# B&R Automation Studio project NAELD004C00R10L518F00 (part 32)

#### Act_Main.st
```iecst
(** 2019-10-30 **)
ACTION Act_Main:

	IF eStatOld <> eStat THEN
		fbInit(bEn := FALSE);
		fbEnt(bEn := FALSE);
		fbPreExit(bEn := FALSE);
		fbExit(bEn := FALSE);
		fbExit1(bEn := FALSE);
		fbStop(bEn := FALSE);
		fbFixClprClampChk(bEn := FALSE);
		fbFixClprUnclampChk(bEn := FALSE);
		fbRmtClprClampChk(bEn := FALSE);
		fbRmtClprUnclampChk(bEn := FALSE);
		fbClprDlyTm(IN := FALSE);

		IF eStatOld <> MagConv2ClpActIdle
			AND eStatOld <> MagConv2ClpActSetMtrSigOnOrLToR
			AND eStatOld <> MagConv2ClpActSetMtrDirOrRToL
			AND eStatOld <> MagConv2ClpActRstMtrSigOnOrLToR
			AND eStatOld <> MagConv2ClpActRstMtrDirOrRToL
			AND eStatOld <> MagConv2ClpActSetMtrAll
			AND eStatOld <> MagConv2ClpActRstMtrAll THEN

			bMtrSigOnOrLToR	:= FALSE;
			bMtrDirOrRToL	:= FALSE;

		END_IF

		usiStep		:= 0;
		usiSubStep	:= 0;
		bReachEnd	:= FALSE;

		sStatTxt	:= a_sStatText[eStat];

		eStatOld	:= eStat;

		eStatus		:= Busy;
	END_IF

	//Main
	CASE eStat OF

		MagConv2ClpActIdle:
			IF EDGENEG(p_bManual) THEN
				bMtrSigOnOrLToR	:= FALSE;
				bMtrDirOrRToL	:= FALSE;
			END_IF

			eStatus	:= Idle;

		MagConv2ClpActInit:
			IF eStatus = Idle OR eStatus = Busy THEN

				eStatus	:= Busy;

				//Magazine Conveyor Init Run
				//Detect Have Magazine
				IF p_bLeftSen OR p_bRightSen THEN
					bHvMag	:= TRUE;
				ELSE
					bHvMag	:= FALSE;
				END_IF

				fbInit.bConvLToR	:= (p_eDirection = ConvDirLToR) OR (p_eDirection = ConvDirLToL);
				fbInit.tTxDlyTm		:= DINT_TO_TIME(p_diInitTm);

				IF fbInit.bConvLToR = TRUE THEN
					fbInit.bEndSen	:= p_bRightSen;
				ELSE
					fbInit.bEndSen	:= p_bLeftSen;
				END_IF

				fbInit(bEn := TRUE);

				bMtrSigOnOrLToR	:= fbInit.bMtrSigOnOrLToR;
				bMtrDirOrRToL	:= fbInit.bMtrDirOrRToL;

				IF fbInit.udiStatus = 0 THEN
					IF fbInit.bConvLToR = TRUE THEN
						IF bHvMag = TRUE AND p_bRightSen = FALSE THEN
							udiStatus	:= 10000;	//Magazine Detected But Not Present At Outlet Sensor (L - R) While Magazine Conveyor Initial
							eStatus		:= Error;
						ELSE
							eStatus	:= Done;
						END_IF
					ELSE
						IF bHvMag = TRUE AND p_bLeftSen = FALSE THEN
							udiStatus	:= 10001;	//Magazine Detected But Not Present At Outlet Sensor (R - L) While Magazine Conveyor Initial
							eStatus		:= Error;
						ELSE
							eStatus	:= Done;
						END_IF
					END_IF
				ELSIF fbInit.udiStatus < 65534 THEN
					udiStatus	:= fbInit.udiStatus;
					eStatus		:= Error;
				END_IF
			END_IF

		MagConv2ClpActInitStopClp:
			IF eStatus = Idle OR eStatus = Busy THEN

				eStatus	:= Busy;

				CASE usiStep OF
					0:	//Unclamp
						bFixClprClampCtrl	:= FALSE;
						bRmtClprClampCtrl	:= FALSE;

						fbFixClprUnclampChk.bExtSen		:= p_bFixClprClampSen;
						fbFixClprUnclampChk.bRetSen		:= p_bFixClprUnclampSen;
						fbFixClprUnclampChk.bRetSafety	:= p_bFixClprUnclampSafetySen;
						fbFixClprUnclampChk(bEn := TRUE);

						fbRmtClprUnclampChk.bExtSen		:= p_bRmtClprClampSen;
						fbRmtClprUnclampChk.bRetSen		:= p_bRmtClprUnclampSen;
						fbRmtClprUnclampChk.bRetSafety	:= p_bRmtClprUnclampSafetySen;
						fbRmtClprUnclampChk(bEn := TRUE);

						IF fbFixClprUnclampChk.udiStatus = 0 AND fbRmtClprUnclampChk.udiStatus = 0 THEN
							usiStep	:= 1;
						ELSIF (fbFixClprUnclampChk.udiStatus > 0 AND fbFixClprUnclampChk.udiStatus < 65534) OR (fbRmtClprUnclampChk.udiStatus > 0 AND fbRmtClprUnclampChk.udiStatus < 65534) THEN
							bFixClprClampCtrl	:= TRUE;
							bRmtClprClampCtrl	:= TRUE;

							eStatus	:= Error;

							IF fbFixClprUnclampChk.udiStatus = 1504 OR fbRmtClprUnclampChk.udiStatus = 1504 THEN
								udiStatus	:= 10002;	//Clamper Clamp Sensor Off Time Out In Unclamp Check While Conveyor Initial With Clamper
							ELSIF fbFixClprUnclampChk.udiStatus = 1505 OR fbRmtClprUnclampChk.udiStatus = 1505 THEN
								udiStatus	:= 10003;	//Clamper Unclamp Sensor On Time Out In Unclamp Check While Conveyor Initial With Clamper
							ELSIF fbFixClprUnclampChk.udiStatus = 1508 OR fbRmtClprUnclampChk.udiStatus = 1508 THEN
								udiStatus	:= 10004;	//Clamper Unclamp Safety Sensor Error In Unclamp Check While Conveyor Initial With Clamper
							ELSE
								IF fbFixClprUnclampChk.udiStatus > 0 AND fbFixClprUnclampChk.udiStatus < 65534 THEN
									udiStatus	:= fbFixClprUnclampChk.udiStatus;
								ELSIF fbRmtClprUnclampChk.udiStatus > 0 AND fbRmtClprUnclampChk.udiStatus < 65534 THEN
									udiStatus	:= fbRmtClprUnclampChk.udiStatus;
								END_IF
							END_IF
						END_IF

					1:	//Magazine Conveyor Init Run
						//Detect Have Magazine
						IF p_bLeftSen OR p_bRightSen THEN
							bHvMag	:= TRUE;
						ELSE
							bHvMag	:= FALSE;
						END_IF

						fbInit.bConvLToR	:= (p_eDirection = ConvDirLToR) OR (p_eDirection = ConvDirLToL);
						fbInit.tTxDlyTm		:= DINT_TO_TIME(p_diInitTm);

						IF fbInit.bConvLToR = TRUE THEN
							fbInit.bEndSen	:= p_bRightSen;
						ELSE
							fbInit.bEndSen	:= p_bLeftSen;
						END_IF

						fbInit(bEn := TRUE);

						bMtrSigOnOrLToR	:= fbInit.bMtrSigOnOrLToR;
						bMtrDirOrRToL	:= fbInit.bMtrDirOrRToL;

						IF fbInit.udiStatus = 0 THEN
							IF fbInit.bConvLToR = TRUE THEN
								IF bHvMag = TRUE AND p_bRightSen = FALSE THEN
									udiStatus	:= 10005;	//Magazine Detected But Not Present At Outlet Sensor (L - R) While Conveyor Initial With Clamper
									eStatus		:= Error;
								ELSE
									usiStep	:= 2;
								END_IF
							ELSE
								IF bHvMag = TRUE AND p_bLeftSen = FALSE THEN
									udiStatus	:= 10006;	//Magazine Detected But Not Present At Outlet Sensor (R - L) While Conveyor Initial With Clamper
									eStatus		:= Error;
								ELSE
									usiStep	:= 2;
								END_IF
							END_IF
						ELSIF fbInit.udiStatus < 65534 THEN
							udiStatus	:= fbInit.udiStatus;
							eStatus		:= Error;
						END_IF

					2:	//Check If Have Magazine
						IF bHvMag = TRUE THEN
							usiStep	:= 4;
						ELSE
							eStatus	:= Done;
						END_IF

					3:	//Fix Clamp
						bFixClprClampCtrl	:= TRUE;

						fbFixClprClampChk.bExtSen		:= p_bFixClprClampSen;
						fbFixClprClampChk.bRetSen		:= p_bFixClprUnclampSen;
						fbFixClprClampChk.bExtSafety	:= p_bFixClprClampSafetySen;
						fbFixClprClampChk(bEn := TRUE);

						IF fbFixClprClampChk.udiStatus = 0 THEN
							//	usiStep	:= 4;
							eStatus	:= Done;
						ELSIF fbFixClprClampChk.udiStatus < 65534 THEN
							bFixClprClampCtrl	:= FALSE;

							eStatus	:= Error;

							IF fbFixClprClampChk.udiStatus = 1503 THEN
								udiStatus	:= 10007;	//Clamper Clamp Sensor On Time Out In Clamp Check While Conveyor Initial With Clamper
							ELSIF fbFixClprClampChk.udiStatus = 1506 THEN
								udiStatus	:= 10008;	//Clamper Unclamp Sensor Off Time Out In Clamp Check While Conveyor Initial With Clamper
							ELSIF fbFixClprClampChk.udiStatus = 1507 THEN
								udiStatus	:= 10009;	//Clamper Clamp Safety Sensor Error In Clamp Check While Conveyor Initial With Clamper
							ELSE
								udiStatus	:= fbFixClprClampChk.udiStatus;
							END_IF
						END_IF

					4:	//Remote Clamp
						bRmtClprClampCtrl	:= TRUE;

						fbRmtClprClampChk.bExtSen		:= p_bRmtClprClampSen;
						fbRmtClprClampChk.bRetSen		:= p_bRmtClprUnclampSen;
						fbRmtClprClampChk.bExtSafety	:= p_bRmtClprClampSafetySen;
						fbRmtClprClampChk(bEn := TRUE);

						IF fbRmtClprClampChk.udiStatus = 0 THEN
							//	eStatus	:= Done;
							usiStep	:= 3;
						ELSIF fbRmtClprClampChk.udiStatus < 65534 THEN
							bRmtClprClampCtrl	:= FALSE;

							eStatus	:= Error;

							IF fbRmtClprClampChk.udiStatus = 1503 THEN
								udiStatus	:= 10007;	//Clamper Clamp Sensor On Time Out In Clamp Check While Conveyor Initial With Clamper
							ELSIF fbRmtClprClampChk.udiStatus = 1506 THEN
								udiStatus	:= 10008;	//Clamper Unclamp Sensor Off Time Out In Clamp Check While Conveyor Initial With Clamper
							ELSIF fbRmtClprClampChk.udiStatus = 1507 THEN
								udiStatus	:= 10009;	//Clamper Clamp Safety Sensor Error In Clamp Check While Conveyor Initial With Clamper
							ELSE
								udiStatus	:= fbRmtClprClampChk.udiStatus;
							END_IF
						END_IF

				END_CASE
			END_IF

		MagConv2ClpActInitClpStop:
			IF eStatus = Idle OR eStatus = Busy THEN

				eStatus	:= Busy;

				CASE usiStep OF
					0:	//Unclamp
						bFixClprClampCtrl	:= FALSE;
						bRmtClprClampCtrl	:= FALSE;

						fbFixClprUnclampChk.bExtSen		:= p_bFixClprClampSen;
						fbFixClprUnclampChk.bRetSen		:= p_bFixClprUnclampSen;
						fbFixClprUnclampChk.bRetSafety	:= p_bFixClprUnclampSafetySen;
						fbFixClprUnclampChk(bEn := TRUE);

						fbRmtClprUnclampChk.bExtSen		:= p_bRmtClprClampSen;
						fbRmtClprUnclampChk.bRetSen		:= p_bRmtClprUnclampSen;
						fbRmtClprUnclampChk.bRetSafety	:= p_bRmtClprUnclampSafetySen;
						fbRmtClprUnclampChk(bEn := TRUE);

						IF fbFixClprUnclampChk.udiStatus = 0 AND fbRmtClprUnclampChk.udiStatus = 0 THEN
							usiStep	:= 1;
						ELSIF (fbFixClprUnclampChk.udiStatus > 0 AND fbFixClprUnclampChk.udiStatus < 65534) OR (fbRmtClprUnclampChk.udiStatus > 0 AND fbRmtClprUnclampChk.udiStatus < 65534) THEN
							bFixClprClampCtrl	:= TRUE;
							bRmtClprClampCtrl	:= TRUE;

							eStatus	:= Error;

							IF fbFixClprUnclampChk.udiStatus = 1504 OR fbRmtClprUnclampChk.udiStatus = 1504 THEN
								udiStatus	:= 10002;	//Clamper Clamp Sensor Off Time Out In Unclamp Check While Conveyor Initial With Clamper
							ELSIF fbFixClprUnclampChk.udiStatus = 1505 OR fbRmtClprUnclampChk.udiStatus = 1505 THEN
								udiStatus	:= 10003;	//Clamper Unclamp Sensor On Time Out In Unclamp Check While Conveyor Initial With Clamper
							ELSIF fbFixClprUnclampChk.udiStatus = 1508 OR fbRmtClprUnclampChk.udiStatus = 1508 THEN
								udiStatus	:= 10004;	//Clamper Unclamp Safety Sensor Error In Unclamp Check While Conveyor Initial With Clamper
							ELSE
								IF fbFixClprUnclampChk.udiStatus > 0 AND fbFixClprUnclampChk.udiStatus < 65534 THEN
									udiStatus	:= fbFixClprUnclampChk.udiStatus;
								ELSIF fbRmtClprUnclampChk.udiStatus > 0 AND fbRmtClprUnclampChk.udiStatus < 65534 THEN
									udiStatus	:= fbRmtClprUnclampChk.udiStatus;
								END_IF
							END_IF
						END_IF

					1:	//Magazine Conveyor Init Run & Clamp
						//Detect Have Magazine
						IF p_bLeftSen OR p_bRightSen THEN
							bHvMag	:= TRUE;
						ELSE
							bHvMag	:= FALSE;
						END_IF

						fbInit.bConvLToR	:= (p_eDirection = ConvDirLToR) OR (p_eDirection = ConvDirLToL);
						fbInit.tTxDlyTm		:= DINT_TO_TIME(p_diInitTm);

						IF fbInit.bConvLToR = TRUE THEN
							fbInit.bEndSen	:= p_bRightSen;
						ELSE
							fbInit.bEndSen	:= p_bLeftSen;
						END_IF

						fbInit(bEn := TRUE);

						bMtrSigOnOrLToR	:= fbInit.bMtrSigOnOrLToR;
						bMtrDirOrRToL	:= fbInit.bMtrDirOrRToL;

						IF fbInit.bEndSen = TRUE THEN
							bReachEnd	:= TRUE;
						END_IF

						IF bReachEnd = TRUE THEN
							fbClprDlyTm(IN := TRUE);
							IF fbClprDlyTm.Q = TRUE THEN
								CASE usiSubStep OF
									//	0:	//Fix Clamp
									//										bFixClprClampCtrl	:= TRUE;

									//										fbFixClprClampChk.bExtSen		:= p_bFixClprClampSen;
									//										fbFixClprClampChk.bRetSen		:= p_bFixClprUnclampSen;
									//										fbFixClprClampChk.bExtSafety	:= p_bFixClprClampSafetySen;
									//										fbFixClprClampChk(bEn := TRUE);
									//
									//										IF fbFixClprClampChk.udiStatus = 0 THEN
									//											usiSubStep	:= 1;
									//										END_IF

									0:	//Remote Clamp
										bRmtClprClampCtrl	:= TRUE;

										fbRmtClprClampChk.bExtSen		:= p_bRmtClprClampSen;
										fbRmtClprClampChk.bRetSen		:= p_bRmtClprUnclampSen;
										fbRmtClprClampChk.bExtSafety	:= p_bRmtClprClampSafetySen;
										fbRmtClprClampChk(bEn := TRUE);

										IF fbRmtClprClampChk.udiStatus = 0 THEN
											usiSubStep	:= 1;
										END_IF

									1:

										bFixClprClampCtrl	:= TRUE;

										fbFixClprClampChk.bExtSen		:= p_bFixClprClampSen;
										fbFixClprClampChk.bRetSen		:= p_bFixClprUnclampSen;
										fbFixClprClampChk.bExtSafety	:= p_bFixClprClampSafetySen;
										fbFixClprClampChk(bEn := TRUE);

								END_CASE
							END_IF
						END_IF

						IF (fbInit.udiStatus = 0) AND ((fbFixClprClampChk.udiStatus = 0 AND fbRmtClprClampChk.udiStatus = 0) OR (bReachEnd = FALSE)) THEN
							IF fbInit.bConvLToR = TRUE THEN
								IF bHvMag = TRUE AND p_bRightSen = FALSE THEN
									udiStatus	:= 10041;	//Magazine Detected But Not Present At Outlet Sensor (L - R) While Conveyor Initial With Clamper
									eStatus		:= Error;
								ELSE
									eStatus		:= Done;
								END_IF
							ELSE
								IF bHvMag = TRUE AND p_bLeftSen = FALSE THEN
									udiStatus	:= 10042;	//Magazine Detected But Not Present At Outlet Sensor (R - L) While Conveyor Initial With Clamper
									eStatus		:= Error;
								ELSE
									eStatus		:= Done;
								END_IF
							END_IF

						ELSIF fbInit.udiStatus > 0 AND fbInit.udiStatus < 65534 THEN
							udiStatus	:= fbInit.udiStatus;
							eStatus		:= Error;

						ELSIF (fbFixClprClampChk.udiStatus > 0 AND fbFixClprClampChk.udiStatus < 65534) OR (fbRmtClprClampChk.udiStatus > 0 AND fbRmtClprClampChk.udiStatus < 65534) THEN
							bFixClprClampCtrl	:= FALSE;
							bRmtClprClampCtrl	:= FALSE;

							eStatus	:= Error;

							IF fbFixClprClampChk.udiStatus = 1503 OR fbRmtClprClampChk.udiStatus = 1503 THEN
								udiStatus	:= 10043;	//Clamper Clamp Sensor On Time Out In Clamp Check While Conveyor Initial With Clamper
							ELSIF fbFixClprClampChk.udiStatus = 1506 OR fbRmtClprClampChk.udiStatus = 1506 THEN
								udiStatus	:= 10044;	//Clamper Unclamp Sensor Off Time Out In Clamp Check While Conveyor Initial With Clamper
							ELSIF fbFixClprClampChk.udiStatus = 1507 OR fbRmtClprClampChk.udiStatus = 1507 THEN
								udiStatus	:= 10045;	//Clamper Clamp Safety Sensor Error In Clamp Check While Conveyor Initial With Clamper
							ELSE
								IF fbFixClprClampChk.udiStatus > 0 AND fbFixClprClampChk.udiStatus < 65534 THEN
									udiStatus	:= fbFixClprClampChk.udiStatus;
								ELSIF fbRmtClprClampChk.udiStatus > 0 AND fbRmtClprClampChk.udiStatus < 65534 THEN
									udiStatus	:= fbRmtClprClampChk.udiStatus;
								END_IF
							END_IF
						END_IF

				END_CASE
			END_IF

		MagConv2ClpActEnt:
			IF eStatus = Idle OR eStatus = Busy THEN

				eStatus	:= Busy;

				//Detect Have Magazine
				IF p_bLeftSen OR p_bRightSen THEN
					bHvMag	:= TRUE;
				END_IF

				//Conveyor Run
				fbEnt.bConvLToR		:= (p_eDirection = ConvDirLToR) OR (p_eDirection = ConvDirLToL);
				fbEnt.tTimeOut		:= DINT_TO_TIME(p_diTxInTimeOut);

				IF fbEnt.bConvLToR = TRUE THEN
					fbEnt.bEndSen	:= p_bRightSen;
				ELSE
					fbEnt.bEndSen	:= p_bLeftSen;
				END_IF

				fbEnt(bEn := TRUE);

				bMtrSigOnOrLToR	:= fbEnt.bMtrSigOnOrLToR;
				bMtrDirOrRToL	:= fbEnt.bMtrDirOrRToL;

				IF fbEnt.udiStatus = 0 THEN
					eStatus		:= Done;
				ELSIF fbEnt.udiStatus < 65534 THEN
					eStatus		:= Error;

					IF fbEnt.udiStatus = 1101 THEN
						udiStatus	:= 10028;	//Transfer In Time Out While Entering Magazine
					ELSE
						udiStatus	:= fbEnt.udiStatus;
					END_IF
				END_IF

			END_IF

		MagConv2ClpActEntStopClp:
			IF eStatus = Idle OR eStatus = Busy THEN

				eStatus	:= Busy;

				CASE usiStep OF
					0:	//Conveyor Enter
						//Detect Have Magazine
						IF p_bLeftSen OR p_bRightSen THEN
							bHvMag	:= TRUE;
						END_IF

						//Conveyor Run
						fbEnt.bConvLToR		:= (p_eDirection = ConvDirLToR) OR (p_eDirection = ConvDirLToL);
						fbEnt.tTimeOut		:= DINT_TO_TIME(p_diTxInTimeOut);

						IF fbEnt.bConvLToR = TRUE THEN
							fbEnt.bEndSen	:= p_bRightSen;
						ELSE
							fbEnt.bEndSen	:= p_bLeftSen;
						END_IF

						fbEnt(bEn := TRUE);

						bMtrSigOnOrLToR	:= fbEnt.bMtrSigOnOrLToR;
						bMtrDirOrRToL	:= fbEnt.bMtrDirOrRToL;

						IF fbEnt.udiStatus = 0 THEN
							usiStep	:= 2;
						ELSIF fbEnt.udiStatus < 65534 THEN
							eStatus	:= Error;

							IF fbEnt.udiStatus = 1101 THEN
								udiStatus	:= 10029;	//Transfer In Time Out While Entering Magazine
							ELSE
								udiStatus	:= fbEnt.udiStatus;
							END_IF
						END_IF

					1:	//Fix Clamp
						bFixClprClampCtrl	:= TRUE;

						fbFixClprClampChk.bExtSen		:= p_bFixClprClampSen;
						fbFixClprClampChk.bRetSen		:= p_bFixClprUnclampSen;
						fbFixClprClampChk.bExtSafety	:= p_bFixClprClampSafetySen;
						fbFixClprClampChk(bEn := TRUE);

						IF fbFixClprClampChk.udiStatus = 0 THEN
							//usiStep	:= 2;
							eStatus	:= Done;
						ELSIF fbFixClprClampChk.udiStatus < 65534 THEN
							bFixClprClampCtrl	:= FALSE;

							eStatus	:= Error;

							IF fbFixClprClampChk.udiStatus = 1503 THEN
								udiStatus	:= 10010;	//Clamper Clamp Sensor On Time Out In Clamp Check While Conveyor Enter With Clamper
							ELSIF fbFixClprClampChk.udiStatus = 1506 THEN
								udiStatus	:= 10011;	//Clamper Unclamp Sensor Off Time Out In Clamp Check While Conveyor Enter With Clamper
							ELSIF fbFixClprClampChk.udiStatus = 1507 THEN
								udiStatus	:= 10012;	//Clamper Clamp Safety Sensor Error In Clamp Check While Conveyor Enter With Clamper
							ELSE
								udiStatus	:= fbFixClprClampChk.udiStatus;
							END_IF
						END_IF

					2:	//Remote Clamp
						bRmtClprClampCtrl	:= TRUE;

						fbRmtClprClampChk.bExtSen		:= p_bRmtClprClampSen;
						fbRmtClprClampChk.bRetSen		:= p_bRmtClprUnclampSen;
						fbRmtClprClampChk.bExtSafety	:= p_bRmtClprClampSafetySen;
						fbRmtClprClampChk(bEn := TRUE);

						IF fbRmtClprClampChk.udiStatus = 0 THEN
							//	eStatus	:= Done;
							usiStep	:= 1;
						ELSIF fbRmtClprClampChk.udiStatus < 65534 THEN
							bRmtClprClampCtrl	:= FALSE;

							eStatus	:= Error;

							IF fbRmtClprClampChk.udiStatus = 1503 THEN
								udiStatus	:= 10010;	//Clamper Clamp Sensor On Time Out In Clamp Check While Conveyor Enter With Clamper
							ELSIF fbRmtClprClampChk.udiStatus = 1506 THEN
								udiStatus	:= 10011;	//Clamper Unclamp Sensor Off Time Out In Clamp Check While Conveyor Enter With Clamper
							ELSIF fbRmtClprClampChk.udiStatus = 1507 THEN
								udiStatus	:= 10012;	//Clamper Clamp Safety Sensor Error In Clamp Check While Conveyor Enter With Clamper
							ELSE
								udiStatus	:= fbRmtClprClampChk.udiStatus;
							END_IF
						END_IF

				END_CASE

			END_IF

		MagConv2ClpActEntClpStop:
			IF eStatus = Idle OR eStatus = Busy THEN

				eStatus	:= Busy;

				//Detect Have Magazine
				IF p_bLeftSen OR p_bRightSen THEN
					bHvMag	:= TRUE;
				END_IF

				//Conveyor Run
				fbEnt.bConvLToR		:= (p_eDirection = ConvDirLToR) OR (p_eDirection = ConvDirLToL);
				fbEnt.tTimeOut		:= DINT_TO_TIME(p_diTxInTimeOut);

				IF fbEnt.bConvLToR = TRUE THEN
					fbEnt.bEndSen	:= p_bRightSen;
				ELSE
					fbEnt.bEndSen	:= p_bLeftSen;
				END_IF

				fbEnt(bEn := TRUE);

				bMtrSigOnOrLToR	:= fbEnt.bMtrSigOnOrLToR;
				bMtrDirOrRToL	:= fbEnt.bMtrDirOrRToL;

				IF fbEnt.bEndSen = TRUE THEN
					bReachEnd	:= TRUE;
				END_IF

				IF bReachEnd = TRUE THEN
					fbClprDlyTm(IN := TRUE);
					IF fbClprDlyTm.Q = TRUE THEN
						CASE usiSubStep OF
							0:	//Fix Clamp
								//								bFixClprClampCtrl	:= TRUE;
								//
								//								fbFixClprClampChk.bExtSen		:= p_bFixClprClampSen;
								//								fbFixClprClampChk.bRetSen		:= p_bFixClprUnclampSen;
								//								fbFixClprClampChk.bExtSafety	:= p_bFixClprClampSafetySen;
								//								fbFixClprClampChk(bEn := TRUE);
								//
								//								IF fbFixClprClampChk.udiStatus = 0 THEN
								//									usiSubStep	:= 1;
								//								END_IF

								bRmtClprClampCtrl	:= TRUE;

								fbRmtClprClampChk.bExtSen		:= p_bRmtClprClampSen;
								fbRmtClprClampChk.bRetSen		:= p_bRmtClprUnclampSen;
								fbRmtClprClampChk.bExtSafety	:= p_bRmtClprClampSafetySen;
								fbRmtClprClampChk(bEn := TRUE);

								IF fbRmtClprClampChk.udiStatus = 0 THEN
									usiSubStep	:= 1;
								END_IF

							1:	//Remote Clamp
								//								bRmtClprClampCtrl	:= TRUE;
								//
								//								fbRmtClprClampChk.bExtSen		:= p_bRmtClprClampSen;
								//								fbRmtClprClampChk.bRetSen		:= p_bRmtClprUnclampSen;
								//								fbRmtClprClampChk.bExtSafety	:= p_bRmtClprClampSafetySen;
								//								fbRmtClprClampChk(bEn := TRUE);

								bFixClprClampCtrl	:= TRUE;

								fbFixClprClampChk.bExtSen		:= p_bFixClprClampSen;
								fbFixClprClampChk.bRetSen		:= p_bFixClprUnclampSen;
								fbFixClprClampChk.bExtSafety	:= p_bFixClprClampSafetySen;
								fbFixClprClampChk(bEn := TRUE);

						END_CASE
					END_IF
				END_IF

				IF fbEnt.udiStatus = 0 AND (fbFixClprClampChk.udiStatus = 0 AND fbRmtClprClampChk.udiStatus = 0) THEN
					eStatus	:= Done;

				ELSIF (fbFixClprClampChk.udiStatus > 0 AND fbFixClprClampChk.udiStatus < 65534) OR (fbRmtClprClampChk.udiStatus > 0 AND fbRmtClprClampChk.udiStatus < 65534) THEN
					bFixClprClampCtrl	:= FALSE;
					bRmtClprClampCtrl	:= FALSE;

					eStatus	:= Error;

					IF fbFixClprClampChk.udiStatus = 1503 OR fbRmtClprClampChk.udiStatus = 1503 THEN
						udiStatus	:= 10034;	//Clamper Clamp Sensor On Time Out In Clamp Check While Conveyor Enter With Clamper
					ELSIF fbFixClprClampChk.udiStatus = 1506 OR fbRmtClprClampChk.udiStatus = 1506 THEN
						udiStatus	:= 10035;	//Clamper Unclamp Sensor Off Time Out In Clamp Check While Conveyor Enter With Clamper
					ELSIF fbFixClprClampChk.udiStatus = 1507 OR fbRmtClprClampChk.udiStatus = 1507 THEN
						udiStatus	:= 10036;	//Clamper Clamp Safety Sensor Error In Clamp Check While Conveyor Enter With Clamper
					ELSE
						IF fbFixClprClampChk.udiStatus > 0 AND fbFixClprClampChk.udiStatus < 65534 THEN
							udiStatus	:= fbFixClprClampChk.udiStatus;
						ELSIF fbRmtClprClampChk.udiStatus > 0 AND fbRmtClprClampChk.udiStatus < 65534 THEN
							udiStatus	:= fbRmtClprClampChk.udiStatus;
						END_IF
					END_IF

				ELSIF fbEnt.udiStatus > 0 AND fbEnt.udiStatus < 65534 THEN
					eStatus	:= Error;

					IF fbEnt.udiStatus = 1101 THEN
						udiStatus	:= 10037;	//Transfer In Time Out While Entering Magazine
					ELSE
						udiStatus	:= fbEnt.udiStatus;
					END_IF

				END_IF

			END_IF

		MagConv2ClpActPreExit:
			IF eStatus = Idle OR eStatus = Busy THEN

				eStatus	:= Busy;

				//Conveyor Run
				fbPreExit.bConvLToR		:= (p_eDirection = ConvDirLToR) OR (p_eDirection = ConvDirRToR);
				fbPreExit.tTxDlyTm		:= DINT_TO_TIME(p_diInitTm);

				IF fbPreExit.bConvLToR = TRUE THEN
					fbPreExit.bEndSen	:= p_bRightSen;
					fbPreExit.bStartSen	:= p_bLeftSen;
				ELSE
					fbPreExit.bEndSen	:= p_bLeftSen;
					fbPreExit.bStartSen	:= p_bRightSen;
				END_IF

				fbPreExit(bEn := TRUE);

				bMtrSigOnOrLToR	:= fbPreExit.bMtrSigOnOrLToR;
				bMtrDirOrRToL	:= fbPreExit.bMtrDirOrRToL;

				IF fbPreExit.udiStatus = 0 THEN
					IF fbPreExit.bEndSen = TRUE THEN
						eStatus	:= Done;
					ELSE
						udiStatus	:= 10046;	//Magazine Not Detected While Pre-Exiting Magazine
						eStatus		:= Error;
					END_IF
				ELSIF fbPreExit.udiStatus < 65534 THEN
					udiStatus	:= fbPreExit.udiStatus;
					eStatus		:= Error;
				END_IF

			END_IF

		MagConv2ClpActPreExitClpr:
			IF eStatus = Idle OR eStatus = Busy THEN

				eStatus	:= Busy;

				CASE usiStep OF
					0:	//Unclamp
						bFixClprClampCtrl	:= FALSE;
						bRmtClprClampCtrl	:= FALSE;

						fbFixClprUnclampChk.bExtSen		:= p_bFixClprClampSen;
						fbFixClprUnclampChk.bRetSen		:= p_bFixClprUnclampSen;
						fbFixClprUnclampChk.bRetSafety	:= p_bFixClprUnclampSafetySen;
						fbFixClprUnclampChk(bEn := TRUE);

						fbRmtClprUnclampChk.bExtSen		:= p_bRmtClprClampSen;
						fbRmtClprUnclampChk.bRetSen		:= p_bRmtClprUnclampSen;
						fbRmtClprUnclampChk.bRetSafety	:= p_bRmtClprUnclampSafetySen;
						fbRmtClprUnclampChk(bEn := TRUE);

						IF fbFixClprUnclampChk.udiStatus = 0 AND fbRmtClprUnclampChk.udiStatus = 0 THEN
							usiStep	:= 1;
						ELSIF (fbFixClprUnclampChk.udiStatus > 0 AND fbFixClprUnclampChk.udiStatus < 65534) OR (fbRmtClprUnclampChk.udiStatus > 0 AND fbRmtClprUnclampChk.udiStatus < 65534) THEN
							bFixClprClampCtrl	:= TRUE;
							bRmtClprClampCtrl	:= TRUE;

							eStatus	:= Error;

							IF fbFixClprUnclampChk.udiStatus = 1504 OR fbRmtClprUnclampChk.udiStatus = 1504 THEN
								udiStatus	:= 10002;	//Clamper Clamp Sensor Off Time Out In Unclamp Check While Conveyor Initial With Clamper
							ELSIF fbFixClprUnclampChk.udiStatus = 1505 OR fbRmtClprUnclampChk.udiStatus = 1505 THEN
								udiStatus	:= 10003;	//Clamper Unclamp Sensor On Time Out In Unclamp Check While Conveyor Initial With Clamper
							ELSIF fbFixClprUnclampChk.udiStatus = 1508 OR fbRmtClprUnclampChk.udiStatus = 1508 THEN
								udiStatus	:= 10004;	//Clamper Unclamp Safety Sensor Error In Unclamp Check While Conveyor Initial With Clamper
							ELSE
								IF fbFixClprUnclampChk.udiStatus > 0 AND fbFixClprUnclampChk.udiStatus < 65534 THEN
									udiStatus	:= fbFixClprUnclampChk.udiStatus;
								ELSIF fbRmtClprUnclampChk.udiStatus > 0 AND fbRmtClprUnclampChk.udiStatus < 65534 THEN
									udiStatus	:= fbRmtClprUnclampChk.udiStatus;
								END_IF
							END_IF
						END_IF

					1:	//Conveyor Pre-Exit
						//Conveyor Run
						fbPreExit.bConvLToR		:= (p_eDirection = ConvDirLToR) OR (p_eDirection = ConvDirRToR);
						fbPreExit.tTxDlyTm		:= DINT_TO_TIME(p_diInitTm);

						IF fbPreExit.bConvLToR = TRUE THEN
							fbPreExit.bEndSen	:= p_bRightSen;
							fbPreExit.bStartSen	:= p_bLeftSen;
						ELSE
							fbPreExit.bEndSen	:= p_bLeftSen;
							fbPreExit.bStartSen	:= p_bRightSen;
						END_IF

						fbPreExit(bEn := TRUE);

						bMtrSigOnOrLToR	:= fbPreExit.bMtrSigOnOrLToR;
						bMtrDirOrRToL	:= fbPreExit.bMtrDirOrRToL;

						IF fbPreExit.udiStatus = 0 THEN
							IF fbPreExit.bEndSen = TRUE THEN
								eStatus	:= Done;
							ELSE
								udiStatus	:= 10046;	//Magazine Not Detected While Pre-Exiting Magazine
								eStatus		:= Error;
							END_IF
						ELSIF fbPreExit.udiStatus < 65534 THEN
							udiStatus	:= fbPreExit.udiStatus;
							eStatus		:= Error;
						END_IF

				END_CASE

			END_IF

		MagConv2ClpActExit:
			IF eStatus = Idle OR eStatus = Busy THEN

				eStatus	:= Busy;

				//Conveyor Run
				fbExit.bConvLToR	:= (p_eDirection = ConvDirLToR) OR (p_eDirection = ConvDirRToR);
				fbExit.tTimeOut		:= DINT_TO_TIME(p_diTxOutTimeOut);

				IF fbExit.bConvLToR = TRUE THEN
					fbExit.bEndSen	:= p_bRightSen;
				ELSE
					fbExit.bEndSen	:= p_bLeftSen;
				END_IF

				fbExit(bEn := TRUE);

				bMtrSigOnOrLToR	:= fbExit.bMtrSigOnOrLToR;
				bMtrDirOrRToL	:= fbExit.bMtrDirOrRToL;

				IF fbExit.udiStatus = 0 THEN
					bHvMag		:= FALSE;
					eStatus		:= Done;
				ELSIF fbExit.udiStatus < 65534 THEN
					eStatus		:= Error;

					IF fbExit.udiStatus = 1101 THEN
						udiStatus	:= 10030;	//Transfer Out Time Out While Exiting Magazine
					ELSE
						udiStatus	:= fbExit.udiStatus;
					END_IF
				END_IF

			END_IF

		MagConv2ClpActExit1:
			IF eStatus = Idle OR eStatus = Busy THEN

				eStatus	:= Busy;

				//Conveyor Run
				fbExit1.bConvLToR		:= (p_eDirection = ConvDirLToR) OR (p_eDirection = ConvDirRToR);
				fbExit1.tTimeOut		:= DINT_TO_TIME(p_diTxOutTimeOut);

				IF fbExit1.bConvLToR = TRUE THEN
					fbExit1.bEndSen	:= p_bRightSen;
				ELSE
					fbExit1.bEndSen	:= p_bLeftSen;
				END_IF

				fbExit1(bEn := TRUE);

				bMtrSigOnOrLToR	:= fbExit1.bMtrSigOnOrLToR;
				bMtrDirOrRToL	:= fbExit1.bMtrDirOrRToL;

				IF fbExit1.udiStatus = 0 THEN
					bHvMag		:= FALSE;
					eStatus		:= Done;
				ELSIF fbExit1.udiStatus < 65534 THEN
					eStatus		:= Error;

					IF fbExit1.udiStatus = 1101 THEN
						udiStatus	:= 10032;	//Transfer Out Time Out While Exiting Magazinie
					ELSE
						udiStatus	:= fbExit1.udiStatus;
					END_IF
				END_IF

			END_IF

		MagConv2ClpActExitClpr:
			IF eStatus = Idle OR eStatus = Busy THEN

				eStatus	:= Busy;

				CASE usiStep OF
					0:	//Unclamp
						bFixClprClampCtrl	:= FALSE;
						bRmtClprClampCtrl	:= FALSE;

						fbFixClprUnclampChk.bExtSen		:= p_bFixClprClampSen;
						fbFixClprUnclampChk.bRetSen		:= p_bFixClprUnclampSen;
						fbFixClprUnclampChk.bRetSafety	:= p_bFixClprUnclampSafetySen;
						fbFixClprUnclampChk(bEn := TRUE);

						fbRmtClprUnclampChk.bExtSen		:= p_bRmtClprClampSen;
						fbRmtClprUnclampChk.bRetSen		:= p_bRmtClprUnclampSen;
						fbRmtClprUnclampChk.bRetSafety	:= p_bRmtClprUnclampSafetySen;
						fbRmtClprUnclampChk(bEn := TRUE);

						IF fbFixClprUnclampChk.udiStatus = 0 AND fbRmtClprUnclampChk.udiStatus = 0 THEN
							usiStep	:= 1;
						ELSIF (fbFixClprUnclampChk.udiStatus > 0 AND fbFixClprUnclampChk.udiStatus < 65534) OR (fbRmtClprUnclampChk.udiStatus > 0 AND fbRmtClprUnclampChk.udiStatus < 65534) THEN
							bFixClprClampCtrl	:= TRUE;
							bRmtClprClampCtrl	:= TRUE;

							eStatus	:= Error;

							IF fbFixClprUnclampChk.udiStatus = 1504 OR fbRmtClprUnclampChk.udiStatus = 1504 THEN
								udiStatus	:= 10002;	//Clamper Clamp Sensor Off Time Out In Unclamp Check While Conveyor Initial With Clamper
							ELSIF fbFixClprUnclampChk.udiStatus = 1505 OR fbRmtClprUnclampChk.udiStatus = 1505 THEN
								udiStatus	:= 10003;	//Clamper Unclamp Sensor On Time Out In Unclamp Check While Conveyor Initial With Clamper
							ELSIF fbFixClprUnclampChk.udiStatus = 1508 OR fbRmtClprUnclampChk.udiStatus = 1508 THEN
								udiStatus	:= 10004;	//Clamper Unclamp Safety Sensor Error In Unclamp Check While Conveyor Initial With Clamper
							ELSE
								IF fbFixClprUnclampChk.udiStatus > 0 AND fbFixClprUnclampChk.udiStatus < 65534 THEN
									udiStatus	:= fbFixClprUnclampChk.udiStatus;
								ELSIF fbRmtClprUnclampChk.udiStatus > 0 AND fbRmtClprUnclampChk.udiStatus < 65534 THEN
									udiStatus	:= fbRmtClprUnclampChk.udiStatus;
								END_IF
							END_IF
						END_IF

					1:	//Conveyor Exit
						//Conveyor Run
						fbExit.bConvLToR	:= (p_eDirection = ConvDirLToR) OR (p_eDirection = ConvDirRToR);
						fbExit.tTimeOut		:= DINT_TO_TIME(p_diTxOutTimeOut);

						IF fbExit.bConvLToR = TRUE THEN
							fbExit.bEndSen	:= p_bRightSen;
						ELSE
							fbExit.bEndSen	:= p_bLeftSen;
						END_IF

						fbExit(bEn := TRUE);

						bMtrSigOnOrLToR	:= fbExit.bMtrSigOnOrLToR;
						bMtrDirOrRToL	:= fbExit.bMtrDirOrRToL;

						IF fbExit.udiStatus = 0 THEN
							bHvMag		:= FALSE;
							eStatus		:= Done;
						ELSIF fbExit.udiStatus < 65534 THEN
							eStatus		:= Error;

							IF fbExit.udiStatus = 1101 THEN
								udiStatus	:= 10031;	//Transfer Out Time Out While Conveyor Exit With Clamper
							ELSE
								udiStatus	:= fbExit.udiStatus;
							END_IF
						END_IF

				END_CASE

			END_IF

		MagConv2ClpActExit1Clpr:
			IF eStatus = Idle OR eStatus = Busy THEN

				eStatus	:= Busy;

				CASE usiStep OF
					0:	//Unclamp
						bFixClprClampCtrl	:= FALSE;
						bRmtClprClampCtrl	:= FALSE;

						fbFixClprUnclampChk.bExtSen		:= p_bFixClprClampSen;
						fbFixClprUnclampChk.bRetSen		:= p_bFixClprUnclampSen;
						fbFixClprUnclampChk.bRetSafety	:= p_bFixClprUnclampSafetySen;
						fbFixClprUnclampChk(bEn := TRUE);

						fbRmtClprUnclampChk.bExtSen		:= p_bRmtClprClampSen;
						fbRmtClprUnclampChk.bRetSen		:= p_bRmtClprUnclampSen;
						fbRmtClprUnclampChk.bRetSafety	:= p_bRmtClprUnclampSafetySen;
						fbRmtClprUnclampChk(bEn := TRUE);

						IF fbFixClprUnclampChk.udiStatus = 0 AND fbRmtClprUnclampChk.udiStatus = 0 THEN
							usiStep	:= 1;
						ELSIF (fbFixClprUnclampChk.udiStatus > 0 AND fbFixClprUnclampChk.udiStatus < 65534) OR (fbRmtClprUnclampChk.udiStatus > 0 AND fbRmtClprUnclampChk.udiStatus < 65534) THEN
							bFixClprClampCtrl	:= TRUE;
							bRmtClprClampCtrl	:= TRUE;

							eStatus	:= Error;

							IF fbFixClprUnclampChk.udiStatus = 1504 OR fbRmtClprUnclampChk.udiStatus = 1504 THEN
								udiStatus	:= 10002;	//Clamper Clamp Sensor Off Time Out In Unclamp Check While Conveyor Initial With Clamper
							ELSIF fbFixClprUnclampChk.udiStatus = 1505 OR fbRmtClprUnclampChk.udiStatus = 1505 THEN
								udiStatus	:= 10003;	//Clamper Unclamp Sensor On Time Out In Unclamp Check While Conveyor Initial With Clamper
							ELSIF fbFixClprUnclampChk.udiStatus = 1508 OR fbRmtClprUnclampChk.udiStatus = 1508 THEN
								udiStatus	:= 10004;	//Clamper Unclamp Safety Sensor Error In Unclamp Check While Conveyor Initial With Clamper
							ELSE
								IF fbFixClprUnclampChk.udiStatus > 0 AND fbFixClprUnclampChk.udiStatus < 65534 THEN
									udiStatus	:= fbFixClprUnclampChk.udiStatus;
								ELSIF fbRmtClprUnclampChk.udiStatus > 0 AND fbRmtClprUnclampChk.udiStatus < 65534 THEN
									udiStatus	:= fbRmtClprUnclampChk.udiStatus;
								END_IF
							END_IF
						END_IF

					1:	//Conveyor Exit
						//Conveyor Run
						fbExit1.bConvLToR		:= (p_eDirection = ConvDirLToR) OR (p_eDirection = ConvDirRToR);
						fbExit1.tTimeOut		:= DINT_TO_TIME(p_diTxOutTimeOut);

						IF fbExit1.bConvLToR = TRUE THEN
							fbExit1.bEndSen	:= p_bRightSen;
						ELSE
							fbExit1.bEndSen	:= p_bLeftSen;
						END_IF

						fbExit1(bEn := TRUE);

						bMtrSigOnOrLToR	:= fbExit1.bMtrSigOnOrLToR;
						bMtrDirOrRToL	:= fbExit1.bMtrDirOrRToL;

						IF fbExit1.udiStatus = 0 THEN
							bHvMag		:= FALSE;
							eStatus		:= Done;
						ELSIF fbExit1.udiStatus < 65534 THEN
							eStatus		:= Error;

							IF fbExit1.udiStatus = 1101 THEN
								udiStatus	:= 10033;	//Transfer Out Time Out While Conveyor Exit With Clamper
							ELSE
								udiStatus	:= fbExit1.udiStatus;
							END_IF
						END_IF

				END_CASE

			END_IF

		MagConv2ClpActFixClprSetAll:
			IF eStatus = Idle OR eStatus = Busy THEN

				eStatus	:= Busy;

				bMtrSigOnOrLToR	:= FALSE;
				bMtrDirOrRToL	:= FALSE;

				bFixClprClampCtrl	:= TRUE;

				eStatus	:= Done;

			END_IF

		MagConv2ClpActFixClprRstAll:
			IF eStatus = Idle OR eStatus = Busy THEN

				eStatus	:= Busy;

				bMtrSigOnOrLToR	:= FALSE;
				bMtrDirOrRToL	:= FALSE;

				bFixClprClampCtrl	:= FALSE;

				eStatus	:= Done;

			END_IF

		MagConv2ClpActFixClprSetClamp:
			IF eStatus = Idle OR eStatus = Busy THEN

				eStatus	:= Busy;

				bMtrSigOnOrLToR	:= FALSE;
				bMtrDirOrRToL	:= FALSE;

				bFixClprClampCtrl	:= TRUE;

				eStatus	:= Done;

			END_IF

		MagConv2ClpActFixClprSetUnclamp:
			IF eStatus = Idle OR eStatus = Busy THEN

				eStatus	:= Busy;

				bMtrSigOnOrLToR	:= FALSE;
				bMtrDirOrRToL	:= FALSE;

				bFixClprClampCtrl	:= FALSE;

				eStatus	:= Done;

			END_IF

		MagConv2ClpActFixClprClamp:
			IF eStatus = Idle OR eStatus = Busy THEN

				eStatus	:= Busy;

				bMtrSigOnOrLToR	:= FALSE;
				bMtrDirOrRToL	:= FALSE;

				bFixClprClampCtrl	:= TRUE;

				fbFixClprClampChk.bExtSen		:= p_bFixClprClampSen;
				fbFixClprClampChk.bRetSen		:= p_bFixClprUnclampSen;
				fbFixClprClampChk.bExtSafety	:= p_bFixClprClampSafetySen;
				fbFixClprClampChk(bEn := TRUE);

				IF fbFixClprClampChk.udiStatus = 0 THEN
					eStatus	:= Done;
				ELSIF fbFixClprClampChk.udiStatus < 65534 THEN
					bFixClprClampCtrl	:= FALSE;

					eStatus	:= Error;

					IF fbFixClprClampChk.udiStatus = 1503 THEN
						udiStatus	:= 10016;	//Clamper Clamp Sensor On Time Out In Clamp Check While Clamper Clamp
					ELSIF fbFixClprClampChk.udiStatus = 1506 THEN
						udiStatus	:= 10017;	//Clamper Unclamp Sensor Off Time Out In Clamp Check While Clamper Clamp
					ELSIF fbFixClprClampChk.udiStatus = 1507 THEN
						udiStatus	:= 10018;	//Clamper Clamp Safety Sensor Error In Clamp Check While Clamper Clamp
					ELSE
						udiStatus	:= fbFixClprClampChk.udiStatus;
					END_IF
				END_IF
			END_IF

		MagConv2ClpActFixClprUnclamp:
			IF eStatus = Idle OR eStatus = Busy THEN

				eStatus	:= Busy;

				bMtrSigOnOrLToR	:= FALSE;
				bMtrDirOrRToL	:= FALSE;

				bFixClprClampCtrl	:= FALSE;

				fbFixClprUnclampChk.bExtSen		:= p_bFixClprClampSen;
				fbFixClprUnclampChk.bRetSen		:= p_bFixClprUnclampSen;
				fbFixClprUnclampChk.bRetSafety	:= p_bFixClprUnclampSafetySen;
				fbFixClprUnclampChk(bEn := TRUE);

				IF fbFixClprUnclampChk.udiStatus = 0 THEN
					eStatus	:= Done;
				ELSIF fbFixClprUnclampChk.udiStatus < 65534 THEN
					bFixClprClampCtrl	:= TRUE;

					eStatus	:= Error;

					IF fbFixClprUnclampChk.udiStatus = 1504 THEN
						udiStatus	:= 10019;	//Clamper Clamp Sensor Off Time Out In Unclamp Check While Clamper Unclamp
					ELSIF fbFixClprUnclampChk.udiStatus = 1505 THEN
						udiStatus	:= 10020;	//Clamper Unclamp Sensor On Time Out In Unclamp Check While Clamper Unclamp
					ELSIF fbFixClprUnclampChk.udiStatus = 1508 THEN
						udiStatus	:= 10021;	//Clamper Unclamp Safety Sensor Error In Unclamp Check While Clamper Unclamp
					ELSE
						udiStatus	:= fbFixClprUnclampChk.udiStatus;
					END_IF
				END_IF

			END_IF

		MagConv2ClpActRmtClprSetAll:
			IF eStatus = Idle OR eStatus = Busy THEN

				eStatus	:= Busy;

				bMtrSigOnOrLToR	:= FALSE;
				bMtrDirOrRToL	:= FALSE;

				bRmtClprClampCtrl	:= TRUE;

				eStatus	:= Done;

			END_IF

		MagConv2ClpActRmtClprRstAll:
			IF eStatus = Idle OR eStatus = Busy THEN

				eStatus	:= Busy;

				bMtrSigOnOrLToR	:= FALSE;
				bMtrDirOrRToL	:= FALSE;

				bRmtClprClampCtrl	:= FALSE;

				eStatus	:= Done;

			END_IF

		MagConv2ClpActRmtClprSetClamp:
			IF eStatus = Idle OR eStatus = Busy THEN

				eStatus	:= Busy;

				bMtrSigOnOrLToR	:= FALSE;
				bMtrDirOrRToL	:= FALSE;

				bRmtClprClampCtrl	:= TRUE;

				eStatus	:= Done;

			END_IF

		MagConv2ClpActRmtClprSetUnclamp:
			IF eStatus = Idle OR eStatus = Busy THEN

				eStatus	:= Busy;

				bMtrSigOnOrLToR	:= FALSE;
				bMtrDirOrRToL	:= FALSE;

				bRmtClprClampCtrl	:= FALSE;

				eStatus	:= Done;

			END_IF

		MagConv2ClpActRmtClprClamp:
			IF eStatus = Idle OR eStatus = Busy THEN

				eStatus	:= Busy;

				bMtrSigOnOrLToR	:= FALSE;
				bMtrDirOrRToL	:= FALSE;

				bRmtClprClampCtrl	:= TRUE;

				fbRmtClprClampChk.bExtSen		:= p_bRmtClprClampSen;
				fbRmtClprClampChk.bRetSen		:= p_bRmtClprUnclampSen;
				fbRmtClprClampChk.bExtSafety	:= p_bRmtClprClampSafetySen;
				fbRmtClprClampChk(bEn := TRUE);

				IF fbRmtClprClampChk.udiStatus = 0 THEN
					eStatus	:= Done;
				ELSIF fbRmtClprClampChk.udiStatus < 65534 THEN
					bRmtClprClampCtrl	:= FALSE;

					eStatus	:= Error;

					IF fbRmtClprClampChk.udiStatus = 1503 THEN
						udiStatus	:= 10016;	//Clamper Clamp Sensor On Time Out In Clamp Check While Clamper Clamp
					ELSIF fbRmtClprClampChk.udiStatus = 1506 THEN
						udiStatus	:= 10017;	//Clamper Unclamp Sensor Off Time Out In Clamp Check While Clamper Clamp
					ELSIF fbRmtClprClampChk.udiStatus = 1507 THEN
						udiStatus	:= 10018;	//Clamper Clamp Safety Sensor Error In Clamp Check While Clamper Clamp
					ELSE
						udiStatus	:= fbRmtClprClampChk.udiStatus;
					END_IF
				END_IF
			END_IF

		MagConv2ClpActRmtClprUnclamp:
			IF eStatus = Idle OR eStatus = Busy THEN

				eStatus	:= Busy;

				bMtrSigOnOrLToR	:= FALSE;
				bMtrDirOrRToL	:= FALSE;

				bRmtClprClampCtrl	:= FALSE;

				fbRmtClprUnclampChk.bExtSen		:= p_bRmtClprClampSen;
				fbRmtClprUnclampChk.bRetSen		:= p_bRmtClprUnclampSen;
				fbRmtClprUnclampChk.bRetSafety	:= p_bRmtClprUnclampSafetySen;
				fbRmtClprUnclampChk(bEn := TRUE);

				IF fbRmtClprUnclampChk.udiStatus = 0 THEN
					eStatus	:= Done;
				ELSIF fbRmtClprUnclampChk.udiStatus < 65534 THEN
					bRmtClprClampCtrl	:= TRUE;

					eStatus	:= Error;

					IF fbRmtClprUnclampChk.udiStatus = 1504 THEN
						udiStatus	:= 10019;	//Clamper Clamp Sensor Off Time Out In Unclamp Check While Clamper Unclamp
					ELSIF fbRmtClprUnclampChk.udiStatus = 1505 THEN
						udiStatus	:= 10020;	//Clamper Unclamp Sensor On Time Out In Unclamp Check While Clamper Unclamp
					ELSIF fbRmtClprUnclampChk.udiStatus = 1508 THEN
						udiStatus	:= 10021;	//Clamper Unclamp Safety Sensor Error In Unclamp Check While Clamper Unclamp
					ELSE
						udiStatus	:= fbRmtClprUnclampChk.udiStatus;
					END_IF
				END_IF

			END_IF

		MagConv2ClpActStop:
			IF eStatus = Idle OR eStatus = Busy THEN

				eStatus	:= Busy;

				//Conveyor Run
				fbStop(bEn := TRUE);

				bMtrSigOnOrLToR	:= fbStop.bMtrSigOnOrLToR;
				bMtrDirOrRToL	:= fbStop.bMtrDirOrRToL;

				IF fbStop.udiStatus = 0 THEN
					eStatus	:= Done;
				ELSIF fbStop.udiStatus < 65534 THEN
					udiStatus	:= fbStop.udiStatus;
					eStatus		:= Error;
				END_IF

			END_IF

		MagConv2ClpActStopClpr:
			IF eStatus = Idle OR eStatus = Busy THEN

				eStatus	:= Busy;

				//Conveyor Run
				fbStop(bEn := TRUE);

				bMtrSigOnOrLToR	:= fbStop.bMtrSigOnOrLToR;
				bMtrDirOrRToL	:= fbStop.bMtrDirOrRToL;

				bFixClprClampCtrl	:= FALSE;
				bRmtClprClampCtrl	:= FALSE;

				fbFixClprUnclampChk.bExtSen		:= p_bFixClprClampSen;
				fbFixClprUnclampChk.bRetSen		:= p_bFixClprUnclampSen;
				fbFixClprUnclampChk.bRetSafety	:= p_bFixClprUnclampSafetySen;
				fbFixClprUnclampChk(bEn := TRUE);

				fbRmtClprUnclampChk.bExtSen		:= p_bRmtClprClampSen;
				fbRmtClprUnclampChk.bRetSen		:= p_bRmtClprUnclampSen;
				fbRmtClprUnclampChk.bRetSafety	:= p_bRmtClprUnclampSafetySen;
				fbRmtClprUnclampChk(bEn := TRUE);

				IF fbStop.udiStatus = 0 AND fbFixClprUnclampChk.udiStatus = 0 AND fbRmtClprUnclampChk.udiStatus = 0 THEN
					eStatus		:= Done;
				ELSIF fbStop.udiStatus > 0 AND fbStop.udiStatus < 65534 THEN
					udiStatus	:= fbStop.udiStatus;
					eStatus		:= Error;
				ELSIF (fbFixClprUnclampChk.udiStatus > 0 AND fbFixClprUnclampChk.udiStatus < 65534) OR (fbRmtClprUnclampChk.udiStatus > 0 AND fbRmtClprUnclampChk.udiStatus < 65534) THEN
					bFixClprClampCtrl	:= TRUE;
					bRmtClprClampCtrl	:= TRUE;

					eStatus	:= Error;

					IF fbFixClprUnclampChk.udiStatus = 1504 OR fbRmtClprUnclampChk.udiStatus = 1504 THEN
						udiStatus	:= 10022;	//Clamper Clamp Sensor Off Time Out In Unclamp Check While Stop With Clamper
					ELSIF fbFixClprUnclampChk.udiStatus = 1505 OR fbRmtClprUnclampChk.udiStatus = 1505 THEN
						udiStatus	:= 10023;	//Clamper Unclamp Sensor On Time Out In Unclamp Check While Stop With Clamper
					ELSIF fbFixClprUnclampChk.udiStatus = 1508 OR fbRmtClprUnclampChk.udiStatus = 1508 THEN
						udiStatus	:= 10024;	//Clamper Unclamp Safety Sensor Error In Unclamp Check While Stop With Clamper
					ELSE
						IF fbFixClprUnclampChk.udiStatus > 0 AND fbFixClprUnclampChk.udiStatus < 65534 THEN
							udiStatus	:= fbFixClprUnclampChk.udiStatus;
						ELSIF fbRmtClprUnclampChk.udiStatus > 0 AND fbRmtClprUnclampChk.udiStatus < 65534 THEN
							udiStatus	:= fbRmtClprUnclampChk.udiStatus;
						END_IF
					END_IF
				END_IF

			END_IF

		MagConv2ClpActSetMtrSigOnOrLToR:
			IF eStatus = Idle OR eStatus = Busy THEN

				bMtrSigOnOrLToR	:= TRUE;

				eStatus	:= Done;

			END_IF

		MagConv2ClpActSetMtrDirOrRToL:
			IF eStatus = Idle OR eStatus = Busy THEN

				bMtrDirOrRToL	:= TRUE;

				eStatus	:= Done;

			END_IF

		MagConv2ClpActRstMtrSigOnOrLToR:
			IF eStatus = Idle OR eStatus = Busy THEN

				bMtrSigOnOrLToR	:= FALSE;

				eStatus	:= Done;

			END_IF

		MagConv2ClpActRstMtrDirOrRToL:
			IF eStatus = Idle OR eStatus = Busy THEN

				bMtrDirOrRToL	:= FALSE;

				eStatus	:= Done;

			END_IF

		MagConv2ClpActSetMtrAll:
			IF eStatus = Idle OR eStatus = Busy THEN

				bMtrSigOnOrLToR	:= TRUE;
				bMtrDirOrRToL	:= TRUE;

				eStatus	:= Done;

			END_IF

		MagConv2ClpActRstMtrAll:
			IF eStatus = Idle OR eStatus = Busy THEN

				bMtrSigOnOrLToR	:= FALSE;
				bMtrDirOrRToL	:= FALSE;

				eStatus	:= Done;

			END_IF

	END_CASE

END_ACTION
```

#### Init.st
```iecst
(** 2019-10-30 **)
PROGRAM _INIT

	(* Always Change If Project Change *)

	//Pass Address To Global Address For External Use
	//Action, State & Status
	p_MagConv2Clp4Stat				:= ADR(eStat);
	p_MagConv2Clp4Status			:= ADR(eStatus);
	p_MagConv2Clp4StatTxt			:= ADR(sStatTxt);

	//Alarm
	p_MagConv2Clp4AlmData			:= ADR(tyAlmData);

	//Output
	p_MagConv2Clp4HvMag				:= ADR(bHvMag);
	p_MagConv2Clp4MtrSigOnOrLToR	:= ADR(bMtrSigOnOrLToR);
	p_MagConv2Clp4MtrDirOrRToL		:= ADR(bMtrDirOrRToL);

	p_MagConv2Clp4FixClprClampCtrl	:= ADR(bFixClprClampCtrl);
	p_MagConv2Clp4RmtClprClampCtrl	:= ADR(bRmtClprClampCtrl);
	p_MagConv2Clp4ClprTwoOutputCtrl	:= ADR(bClprTwoOutputControl);

	(* Always Change If Project Change *)

END_PROGRAM
```

### Program Logical/CANOpenServo/AW/AWOpen

#### InputRef.var
```iecst
(*2020-05-26*)
(**)
(*General*)
VAR
	p_eAct : REFERENCE TO eAWAction;
	p_udiRstErr : REFERENCE TO UDINT;
	p_bPrep : REFERENCE TO BOOL;
	p_bEn : REFERENCE TO BOOL;
	p_bDis : REFERENCE TO BOOL;
END_VAR
(**)
(*Configuration*)
VAR
	p_bOps : REFERENCE TO BOOL;
	p_bManual : REFERENCE TO BOOL;
	p_diWidthAtHmPos : REFERENCE TO DINT;
	p_tyTuning : REFERENCE TO tyMotionCANTuning;
	p_diGoWidth : REFERENCE TO DINT;
	p_diJogVelInUMPS : REFERENCE TO DINT;
	p_diMovePosInUM : REFERENCE TO DINT;
	p_diMoveDistInUM : REFERENCE TO DINT;
	p_diMoveVelInUMPS : REFERENCE TO DINT;
	p_diMoveAcc : REFERENCE TO DINT;
	p_diMoveDec : REFERENCE TO DINT;
	p_diMinAbsPosInUM : REFERENCE TO DINT;
	p_diMaxAbsPosInUM : REFERENCE TO DINT;
	p_diMinWidthInUM : REFERENCE TO DINT;
	p_diMaxWidthInUM : REFERENCE TO DINT;
	p_diWidthOffsetInUM : REFERENCE TO DINT;
	p_bInletSensor : REFERENCE TO BOOL;
	p_bOutletSensor : REFERENCE TO BOOL;
	p_bClearSensor : REFERENCE TO BOOL;
	p_bMiddleSensor : REFERENCE TO BOOL;
	p_bInterruptSensor : REFERENCE TO BOOL;
	p_bOpenInterruptSensor : REFERENCE TO BOOL;
	p_bCloseInterruptSensor : REFERENCE TO BOOL;
	p_bSafetyInterruptSen : REFERENCE TO BOOL;
	p_bDir : REFERENCE TO BOOL;
	p_bDirBl : REFERENCE TO BOOL;
	p_bNoIndexPulse : REFERENCE TO BOOL;
	p_usiNode : REFERENCE TO USINT;
	p_sDevice : REFERENCE TO STRING[3];
	p_sProgNm : REFERENCE TO STRING[15];
	p_diMoveBacklashDistInUM : REFERENCE TO DINT;
	p_diPitchInUM : REFERENCE TO DINT;
	p_tyParamInHm : REFERENCE TO tyMotionCANParamInHm;
	p_tyParamInConvert : REFERENCE TO tyMotionCANParamInConvert;
	p_bNtSettingsLoadDone : REFERENCE TO BOOL;
	p_bOpsAWStepMove : REFERENCE TO BOOL;
	p_eNtParamMotorType : REFERENCE TO eServoMotorType;
	p_bUITeachServo : REFERENCE TO BOOL;
	p_bOutletShutterCloseRS : REFERENCE TO BOOL;
	p_bProjInletShutPrep : REFERENCE TO BOOL;
	p_bProjOutletShutPrep : REFERENCE TO BOOL;
	p_bOutShutterDis : REFERENCE TO BOOL;
	p_bInletShutterCloseRS : REFERENCE TO BOOL;
	p_bPullerExtSen : REFERENCE TO BOOL;
	p_bPullerRetSen : REFERENCE TO BOOL;
	p_eTravLifPosGo : REFERENCE TO eTravLifLDPos;
END_VAR
```

#### InputRef_Link.var
```iecst
(*2019-04-09*)
(**)
(*External Data*)
VAR
	p_bLinkOpsRun : REFERENCE TO BOOL;
	p_bLinkStartupRun : REFERENCE TO BOOL;
END_VAR
(**)
VAR
	p_eLinkMag : REFERENCE TO eLDMag;
	p_usiLinkMod : REFERENCE TO USINT;
	p_eLinkTravAct : REFERENCE TO eTravAction;
	p_bLinkSafetyRelay : REFERENCE TO BOOL;
	p_bNtParamAutoRcpPrep : REFERENCE TO BOOL;
	p_bHermesSvyPrep : REFERENCE TO BOOL;
	p_bMcParamHermesSvyEn : REFERENCE TO BOOL;
	p_eNtParamCustomerReq : REFERENCE TO eCustomer;
	p_bMcParamMesRFIDEn : REFERENCE TO BOOL;
END_VAR
```

#### Local.var
```iecst
(*2020-05-26*)
(**)
(*Local Action, State & Status*)
VAR
	eAct : eAWAction := AWActIdle;
	eStat : eAWAction := AWActIdle;
	eMainStatus : eFBStatus := Idle;
	eStatus : eFBStatus := Idle;
	eStatus1 : eFBStatus := Idle;
	eStatus2 : eFBStatus := Idle;
	eStatus3 : eFBStatus := Idle;
	udiStatus : UDINT := 0;
	udiStatus1 : UDINT := 0;
	udiStatus2 : UDINT := 0;
	udiStatus3 : UDINT := 0;
	sStatTxt : STRING[200] := '';
	a_sStatText : ARRAY[0..50] OF STRING[200] := ['Idling','Going Width','Full Homing','Powering On','Powering Off','Homing','Moving Absolute','Moving Relative','Jogging Open','Jogging Close','Jogging Stop','Resetting Axis Error','Stopping','Writing SDO','Background Starting Module OK Check','Background Stopping Module OK Check','Going Width And Power Off','Reset Servo Module Node',33('')];
END_VAR
(**)
(*Local Alarm*)
VAR
	tyAlmData : tyAlmDat;
	tyAlmData1 : tyAlmDat;
	tyAlmData2 : tyAlmDat;
	tyAlmData3 : tyAlmDat;
	a_tyAlmText : ARRAY[10000..10299] OF tyAlmTxt := [(sAlmText:='Axis Move Abnormally By External Force',sRcyText:='Servo Motor Abnormal Operation. Reset And Resume Operation. If The Problem Persists, Please Contact Nutek For A Possible Solution.'),(sAlmText:='CANOpen Communication Error, ModuleOK Not TRUE',sRcyText:='Fail While Read/Write Data. Reset The Error And Resume Operation.'),(sAlmText:='Power On Time Out While Going New Width',sRcyText:='Timeout Expired Before Operation Completed. Reset And Resume Operation.'),(sAlmText:='Homing Time Out While Going New Width',sRcyText:='Timeout Expired Before Operation Completed. Reset And Resume Operation.'),(sAlmText:='Move Absolute Time Out While Going New Width',sRcyText:='Timeout Expired Before Operation Completed. Reset And Resume Operation.'),(sAlmText:='Stop Motion Time Out While Going New Width',sRcyText:='Timeout Expired Before Operation Completed. Reset And Resume Operation.'),(sAlmText:='Axis Error Reset Failed While Going New Width',sRcyText:='Axis Error Reset Failed. Please Retry Again Reset Operation. If The Problem Persists, Please Contact Nutek For A Possible Solution.'),(sAlmText:='Axis Error Occur In Move Absolute While Going New Width',sRcyText:='Servo Motor Abnormal Operation. Reset And Resume Operation. If The Problem Persists, Please Contact Nutek For A Possible Solution.'),(sAlmText:='Axis Error Occur In Homing While Going New Width',sRcyText:='Servo Motor Abnormal Operation. Reset And Resume Operation. If The Problem Persists, Please Contact Nutek For A Possible Solution.'),(sAlmText:='Homing Done But Home Flag Is Not Activated While Going New Width',sRcyText:='Servo Motor Abnormal Operation. Reset And Resume Operation. If The Problem Persists, Please Contact Nutek For A Possible Solution.'),(sAlmText:='Forward Limit Activated In Homing While Going New Width',sRcyText:='Forward Limit Switch Is Activated. Reset The Error By Operate The Motor Backwards.'),(sAlmText:='Reverse Limit Activated In Homing While Going New Width',sRcyText:='Reverse Limit Switch Is Activated. Reset The Error By Operate The Motor Backwards.'),(sAlmText:='Forward Limit Activated In Move Absolute While Going New Width',sRcyText:='Forward Limit Switch Is Activated. Reset The Error By Operate The Motor Backwards.'),(sAlmText:='Reverse Limit Activated In Move Absolute While Going New Width',sRcyText:='Reverse Limit Switch Is Activated. Reset The Error By Operate The Motor Backwards.'),(sAlmText:='Power On Time Out While Full Homing',sRcyText:='Timeout Expired Before Operation Completed. Reset And Resume Operation.'),(sAlmText:='Homing Time Out While Full Homing',sRcyText:='Timeout Expired Before Operation Completed. Reset And Resume Operation.'),(sAlmText:='Stop Motion Time Out While Full Homing',sRcyText:='Timeout Expired Before Operation Completed. Reset And Resume Operation.'),(sAlmText:='Axis Error Reset Failed While Full Homing',sRcyText:='Axis Error Reset Failed. Please Retry Again Reset Operation. If The Problem Persists, Please Contact Nutek For A Possible Solution.'),(sAlmText:='Axis Error Occur In Homing While Full Homing',sRcyText:='Servo Motor Abnormal Operation. Reset And Resume Operation. If The Problem Persists, Please Contact Nutek For A Possible Solution.'),(sAlmText:='Homing Done But Home Flag Is Not Activated While Full Homing',sRcyText:='Servo Motor Abnormal Operation. Reset And Resume Operation. If The Problem Persists, Please Contact Nutek For A Possible Solution.'),(sAlmText:='Forward Limit Activated In Homing While Full Homing',sRcyText:='Forward Limit Switch Is Activated. Reset The Error By Operate The Motor Backwards.'),(sAlmText:='Reverse Limit Activated In Homing While Full Homing',sRcyText:='Reverse Limit Switch Is Activated. Reset The Error By Operate The Motor Backwards.'),(sAlmText:='Power On Time Out',sRcyText:='Timeout Expired Before Operation Completed. Reset And Resume Operation.'),(sAlmText:='Power Off Time Out',sRcyText:='Timeout Expired Before Operation Completed. Reset And Resume Operation.'),(sAlmText:='Homing Time Out',sRcyText:='Timeout Expired Before Operation Completed. Reset And Resume Operation.'),(sAlmText:='Move Absolute Time Out',sRcyText:='Timeout Expired Before Operation Completed. Reset And Resume Operation.'),(sAlmText:='Move Relative Time Out',sRcyText:='Timeout Expired Before Operation Completed. Reset And Resume Operation.'),(sAlmText:='Stop Motion Time Out',sRcyText:='Timeout Expired Before Operation Completed. Reset And Resume Operation.'),(sAlmText:='SDO Write Error',sRcyText:='Fail While Write Data. Reset The Error And Resume Operation.'),(sAlmText:='Request Absolute Position Out Of Range',sRcyText:='Request Absolute Position Does Not Fall Within The Expected Range.'),(sAlmText:='Inlet Sensor Interrupt Auto Width Movement',sRcyText:='Operation Stop Due To The Interruption Of Sensor While Auto Width Moving. Solve The Interruption To Resume Operation.'),(sAlmText:='Outlet Sensor Interrupt Auto Width Movement',sRcyText:='Operation Stop Due To The Interruption Of Sensor While Auto Width Moving. Solve The Interruption To Resume Operation.'),(sAlmText:='Clear Sensor Interrupt Auto Width Movement',sRcyText:='Operation Stop Due To The Interruption Of Sensor While Auto Width Moving. Solve The Interruption To Resume Operation.'),(sAlmText:='Middle Sensor Interrupt Auto Width Movement',sRcyText:='Operation Stop Due To The Interruption Of Sensor While Auto Width Moving. Solve The Interruption To Resume Operation.'),(sAlmText:='Sensor Interrupt Auto Width Movement',sRcyText:='Operation Stop Due To The Interruption Of Sensor While Auto Width Moving. Solve The Interruption To Resume Operation.'),(sAlmText:='Power On Time Out While Going New Width And Off',sRcyText:='Timeout Expired Before Operation Completed. Reset And Resume Operation.'),(sAlmText:='Homing Time Out While Going New Width And Off',sRcyText:='Timeout Expired Before Operation Completed. Reset And Resume Operation.'),(sAlmText:='Move Absolute Time Out While Going New Width And Off',sRcyText:='Timeout Expired Before Operation Completed. Reset And Resume Operation.'),(sAlmText:='Stop Motion Time Out While Going New Width And Off',sRcyText:='Timeout Expired Before Operation Completed. Reset And Resume Operation.'),(sAlmText:='Axis Error Reset Failed While Going New Width And Off',sRcyText:='Axis Error Reset Failed. Please Retry Again Reset Operation. If The Problem Persists, Please Contact Nutek For A Possible Solution.'),(sAlmText:='Axis Error Occur In Move Absolute While Going New Width And Off',sRcyText:='Servo Motor Abnormal Operation. Reset And Resume Operation. If The Problem Persists, Please Contact Nutek For A Possible Solution.'),(sAlmText:='Axis Error Occur In Homing While Going New Width And Off',sRcyText:='Servo Motor Abnormal Operation. Reset And Resume Operation. If The Problem Persists, Please Contact Nutek For A Possible Solution.'),(sAlmText:='Homing Done But Home Flag Is Not Activated While Going New Width And Off',sRcyText:='Servo Motor Abnormal Operation. Reset And Resume Operation. If The Problem Persists, Please Contact Nutek For A Possible Solution.'),(sAlmText:='Forward Limit Activated In Homing While Going New Width And Off',sRcyText:='Forward Limit Switch Is Activated. Reset The Error By Operate The Motor Backwards.'),(sAlmText:='Reverse Limit Activated In Homing While Going New Width And Off',sRcyText:='Reverse Limit Switch Is Activated. Reset The Error By Operate The Motor Backwards.'),(sAlmText:='Forward Limit Activated In Move Absolute While Going New Width And Off',sRcyText:='Forward Limit Switch Is Activated. Reset The Error By Operate The Motor Backwards.'),(sAlmText:='Reverse Limit Activated In Move Absolute While Going New Width And Off',sRcyText:='Reverse Limit Switch Is Activated. Reset The Error By Operate The Motor Backwards.'),2((sAlmText:='Sensor Interrupt Auto Width Movement',sRcyText:='Operation Stop Due To The Interruption Of Sensor While Auto Width Moving. Solve The Interruption To Resume Operation.')),249((0)),(sAlmText:='Forward Limit Activated',sRcyText:='Forward Limit Switch Is Activated. Reset The Error By Operate The Motor Backwards.'),(sAlmText:='Reverse Limit Activated',sRcyText:='Reverse Limit Switch Is Activated. Reset The Error By Operate The Motor Backwards.')];
END_VAR
(**)
(*Local Output*)
VAR
	tyParamOut : tyMotionCANParamOut;
	sAxisErrTxt : STRING[80];
	bWidthPosDiff : BOOL;
	bJogOpen : BOOL;
	bJogClose : BOOL;
	bJogging : BOOL;
	bOpenSen : BOOL;
	bCloseSen : BOOL;
END_VAR
(**)
(*Local Input*)
VAR
	udiRstErr : UDINT := 0;
	bPrep : BOOL := TRUE;
	bEn : BOOL := TRUE;
	bDis : BOOL := FALSE;
	bOps : BOOL := FALSE;
	bManual : BOOL := FALSE;
	diWidthAtHmPos : DINT := 400;
	tyTuning : tyMotionCANTuning;
	diGoWidth : DINT := 100000;
	diJogVelInUMPS : DINT := 10000;
	diMovePosInUM : DINT := 0;
	diMoveDistInUM : DINT := 0;
	diMoveVelInUMPS : DINT := 10000;
	diMoveAcc : DINT := 500;
	diMoveDec : DINT := 500;
	diMinAbsPosInUM : DINT := -3000;
	diMaxAbsPosInUM : DINT := 10000000;
	diMinWidthInUM : DINT := 70000;
	diMaxWidthInUM : DINT := 460000;
	diWidthOffsetInUM : DINT := 0;
	bInletSensor : BOOL;
	bOutletSensor : BOOL;
	bClearSensor : BOOL;
	bMiddleSensor : BOOL;
	bInterruptSensor : BOOL;
	bOpenInterruptSensor : BOOL;
	bCloseInterruptSensor : BOOL;
	bDir : BOOL;
	bDirBl : BOOL;
	bNoIndexPulse : BOOL;
	usiNode : USINT;
	sDevice : STRING[3];
	sProgNm : STRING[15] := 'AWOpen';
	diMoveBacklashDistInUM : DINT := 3000;
	diPitchInUM : DINT := 3000;
	tyParamInHm : tyMotionCANParamInHm;
	tyParamInConvert : tyMotionCANParamInConvert := (diPitchInUM:=3000);
	bNtSettingsLoadDone : BOOL := TRUE;
	eMotorType : eServoMotorType := DeltaAsdaA2;
END_VAR
(**)
(*Local*)
VAR
	bRstErr : BOOL;
	udiRstErrOld : UDINT;
	bInitDone : BOOL;
	bInitialDone : BOOL;
	bModuleOKChk : BOOL := TRUE;
	bModuleOK : BOOL;
	bModuleNotOK : BOOL := TRUE;
	bModuleNotOKLock : BOOL;
	bNotInterruptible : BOOL;
	bInterruptSensor1 : BOOL;
	bInterruptSensor2 : BOOL;
	diActualPosInUMOld : DINT;
	usiRstStep : USINT := 0;
	usiStep : USINT;
	usiCount : USINT;
	fbTm : TON := (PT:=T#2s);
	fbServoModuleNotOk : TON := (IN:=FALSE,PT:=T#2s);
	fbServoModuleOk : TON := (IN:=FALSE,PT:=T#5s);
	fbRstNodeTimer : TON := (PT:=T#3s);
	tyParamInMove : tyMotionCANParamInMove;
	tyParamInDriver : tyMotionCANDriverIn;
	tyParamOutDriver : tyMotionCANDriverOut := (siModOfOpt_6060:=6);
	fbStop : fbMotionCANStop;
	fbRstAxisErr : fbMotionCANRstAxisErr;
	fbJog : fbMotionCANJog;
	fbMovRel : fbMotionCANMovRel;
	fbMovAbs : fbMotionCANMovAbs;
	fbHoming : fbMotionCANHoming;
	fbPwrOff : fbMotionCANPwrOff;
	fbPwrOn : fbMotionCANPwrOn;
	fbFullHm : fbMotionCANFullHm;
	fbFullMovAbs : fbMotionCANFullMovAbs;
	fbFullMovAbsBl : fbMotionCANFullMovAbsBl;
	fbModuleOK : fbMotionCANModuleOK;
	fbSDOWrite : fbCANSDOWriteArrayParam;
	udiModuleNum : UDINT := 1;
END_VAR
```

#### Act_Alarm1.st
```iecst
(** 2020-03-16 **)
ACTION Act_Alarm1:

	//Error
	IF EDGEPOS(eStatus1 = Error) THEN

		tyAlmData1.sProgNm		:= p_sProgNm;
		tyAlmData1.udiCode		:= udiStatus1;
		tyAlmData1.eSeverity	:= AlmSeverityError;
		tyAlmData1.udiRunTime	:= tyAlmData1.udiRunTime + 1;
		tyAlmData1.bAlm			:= TRUE;
		tyAlmData1.udiModuleNum  := udiModuleNum;
		g_sAWOpenProgNm			:= p_sProgNm;
		//Get Error Message
		IF tyAlmData1.udiCode < 10000 OR tyAlmData1.udiCode > 10099 THEN
			tyAlmData1.sAlmMsg	:= 'Unknown';
			tyAlmData1.sRcyMsg	:= 'Unknown';
		ELSE
			tyAlmData1.sAlmMsg	:= a_tyAlmText[tyAlmData1.udiCode].sAlmText;
			tyAlmData1.sRcyMsg	:= a_tyAlmText[tyAlmData1.udiCode].sRcyText;
		END_IF

		sStatTxt	:= tyAlmData1.sAlmMsg;

	ELSIF bRstErr AND (tyAlmData1.udiCode <> 0) THEN

		tyAlmData1.udiCode		:= 0;
		tyAlmData1.eSeverity	:= AlmSeverityNA;
		tyAlmData1.sAlmMsg		:= '';
		tyAlmData1.sRcyMsg		:= '';
		tyAlmData1.bAlm			:= FALSE;

		sStatTxt	:= a_sStatText[eStat];

	END_IF

END_ACTION
```

#### Act_Alarm2.st
```iecst
(** 2020-03-16 **)
ACTION Act_Alarm2:

	//Error
	IF EDGEPOS(eStatus2 = Error) THEN

		tyAlmData2.sProgNm		:= p_sProgNm;
		tyAlmData2.udiCode		:= udiStatus2;
		tyAlmData2.eSeverity	:= AlmSeverityError;
		tyAlmData2.udiRunTime	:= tyAlmData2.udiRunTime + 1;
		tyAlmData2.bAlm			:= TRUE;
		tyAlmData2.udiModuleNum  := udiModuleNum;
		g_sAWOpenProgNm			:= p_sProgNm;
		//Get Error Message
		IF tyAlmData2.udiCode < 10000 OR tyAlmData2.udiCode > 10099 THEN
			tyAlmData2.sAlmMsg	:= 'Unknown';
			tyAlmData2.sRcyMsg	:= 'Unknown';
		ELSE
			tyAlmData2.sAlmMsg	:= a_tyAlmText[tyAlmData2.udiCode].sAlmText;
			tyAlmData2.sRcyMsg	:= a_tyAlmText[tyAlmData2.udiCode].sRcyText;
		END_IF

		sStatTxt	:= tyAlmData2.sAlmMsg;

	ELSIF bRstErr AND (tyAlmData2.udiCode <> 0) THEN

		tyAlmData2.udiCode		:= 0;
		tyAlmData2.eSeverity	:= AlmSeverityNA;
		tyAlmData2.sAlmMsg		:= '';
		tyAlmData2.sRcyMsg		:= '';
		tyAlmData2.bAlm			:= FALSE;

		sStatTxt	:= a_sStatText[eStat];

	END_IF

END_ACTION
```

#### Act_Alarm3.st
```iecst
(** 2020-03-16 **)
ACTION Act_Alarm3:

	//Error
	IF EDGEPOS(eStatus3 = Error) THEN

		tyAlmData3.sProgNm		:= p_sProgNm;
		tyAlmData3.udiCode		:= udiStatus3;
		tyAlmData3.eSeverity	:= AlmSeverityError;
		tyAlmData3.udiRunTime	:= tyAlmData3.udiRunTime + 1;
		tyAlmData3.bAlm			:= TRUE;
		tyAlmData3.udiModuleNum  := udiModuleNum;
		g_sAWOpenProgNm			:= p_sProgNm;
		//Get Error Message
		IF tyAlmData3.udiCode < 10000 OR tyAlmData3.udiCode > 10099 THEN
			tyAlmData3.sAlmMsg	:= 'Unknown';
			tyAlmData3.sRcyMsg	:= 'Unknown';
		ELSE
			tyAlmData3.sAlmMsg	:= a_tyAlmText[tyAlmData3.udiCode].sAlmText;
			tyAlmData3.sRcyMsg	:= a_tyAlmText[tyAlmData3.udiCode].sRcyText;
		END_IF

		sStatTxt	:= tyAlmData3.sAlmMsg;

	ELSIF bRstErr AND (tyAlmData3.udiCode <> 0) THEN

		tyAlmData3.udiCode		:= 0;
		tyAlmData3.eSeverity	:= AlmSeverityNA;
		tyAlmData3.sAlmMsg		:= '';
		tyAlmData3.sRcyMsg		:= '';
		tyAlmData3.bAlm			:= FALSE;

		sStatTxt	:= a_sStatText[eStat];

	END_IF

END_ACTION
```

#### Act_Background.st
```iecst
(** 2020-05-26 **)
ACTION Act_Background:

	//Update Parameter
	IF bModuleOK = TRUE THEN

		tyParamInMove.diPosInUM		:= p_diMovePosInUM;
		tyParamInMove.diDistInUM	:= p_diMoveDistInUM;
		tyParamInMove.diVelInUMPS	:= p_diMoveVelInUMPS;
		tyParamInMove.diAcc			:= p_diMoveAcc;
		tyParamInMove.diDec			:= p_diMoveDec;

		fMotionCANUpdtDat(ADR(tyParamOut) , p_tyParamInConvert , tyParamOutDriver , tyParamInDriver , tyParamInMove , p_tyParamInHm , p_bDir, p_eNtParamMotorType);

		bWidthPosDiff	:= (tyParamOut.bIsHomed = FALSE) OR ((ABS((fAWWidthToPosInUM(p_diGoWidth , p_diWidthAtHmPos)) - tyParamOut.diActualPosInUM)) > 500);

		p_tyParamInConvert.diPitchInUM	:= fPitchCalc(p_diWidthOffsetInUM , p_diMaxWidthInUM , p_diMinWidthInUM , p_diPitchInUM);

		fbFullMovAbsBl.tyParamInConvert					:= p_tyParamInConvert;

		IF p_bDir = TRUE THEN
			bOpenSen	:= tyParamOut.bFwdLmtSen;
			bCloseSen	:= tyParamOut.bRevLmtSen;
		ELSE
			bOpenSen	:= tyParamOut.bRevLmtSen;
			bCloseSen	:= tyParamOut.bFwdLmtSen;
		END_IF

		CASE p_eNtParamMotorType OF
			DeltaAsdaA2:
				CASE tyParamOut.udiAxisErrID OF
					8976:	sAxisErrTxt	:= 'Over Current';
					12560:	sAxisErrTxt	:= 'Over Voltage';
					12576:	sAxisErrTxt	:= 'Under Voltage';
					12592:	sAxisErrTxt	:= 'Input Power Phase Loss';
					12816:	sAxisErrTxt	:= 'Regeneration Error';
					12848:	sAxisErrTxt	:= 'Overload';
					12849:	sAxisErrTxt	:= 'Pre-overload Warning';
					13056:	sAxisErrTxt	:= 'U,V,W Wiring Error';
					16912:	sAxisErrTxt	:= 'IGBT Temperature Error';
					21296:	sAxisErrTxt	:= 'Memory Error';
					21569:	sAxisErrTxt	:= 'Emergency Stop Activated';
					21570:	sAxisErrTxt	:= 'Forward Limit Switch Error';
					21571:	sAxisErrTxt	:= 'Reverse Limit Switch Error';
					21572:	sAxisErrTxt	:= 'Forward Software Limit';
					21573:	sAxisErrTxt	:= 'Reverse Software Limit';
					21760:	sAxisErrTxt	:= 'DSP Firmware Upgrade';
					25088:	sAxisErrTxt	:= 'CANopen SYNC Error';
					25360:	sAxisErrTxt	:= 'CANopen Data Initial Error';
					25376:	sAxisErrTxt	:= 'Adjustment Error';
					28961:	sAxisErrTxt	:= 'Motor Protection Error';
					28962:	sAxisErrTxt	:= 'Motor Error';
					29445:	sAxisErrTxt	:= 'Encoder Error';
					29446:	sAxisErrTxt	:= 'Encoder Output Error';
					29968:	sAxisErrTxt	:= 'Serial Communication Error';
					29984:	sAxisErrTxt	:= 'Serial Communication Time Out';
					33024:	sAxisErrTxt	:= 'CANbus Error (Bus-off)';
					33040:	sAxisErrTxt	:= 'CANopen SDO receive buffer overrun';
					33056:	sAxisErrTxt	:= 'CANbus Error (Warning)';
					33072:	sAxisErrTxt	:= 'Node Guarding or Heartbeat Error';
					33280:	sAxisErrTxt	:= 'CANopen PDO Object Error';
					33792:	sAxisErrTxt	:= 'Over Speed';
					34304:	sAxisErrTxt	:= 'Abnormal Pulse Control Command';
					34320:	sAxisErrTxt	:= 'Full Closed Loop Excessive Deviation';
					34321:	sAxisErrTxt	:= 'Excessive Deviation';
				END_CASE

			SchneiderLexium28:
				CASE tyParamOut.udiAxisErrID OF
					8724:	sAxisErrTxt	:= 'Over Current';
					8976:	sAxisErrTxt	:= 'Motor Overload';
					8977:	sAxisErrTxt	:= 'Drive overload (foldback)';
					9088:	sAxisErrTxt	:= 'Calculated offsets for current sensors out OF range';
					9089:	sAxisErrTxt := 'Motor phase missing';
					9090:	sAxisErrTxt := 'Overcurrent detected at one OF the digital outputs';
					12560:	sAxisErrTxt	:= 'DC Bus Over Voltage';
					12576:	sAxisErrTxt	:= 'DC Bus Under Voltage';
					12672:	sAxisErrTxt	:= 'Braking Resistor Overload';
					12673:	sAxisErrTxt	:= 'Safety function Safe Torque Off (STO) triggered';
					12674:	sAxisErrTxt	:= 'DC bus voltage measurement';
					12675:	sAxisErrTxt	:= 'Missing mains supply, undervoltage mains supply';
					12676:	sAxisErrTxt := 'The encoder supply voltage has dropped under operational value';
					12677:	sAxisErrTxt := 'The multi turn encoder battery voltage has dropped under 3 Vdc';
					12678:	sAxisErrTxt := 'Internal position synchronization error	detected between the multi turn AND the single turn modules';
					12679:	sAxisErrTxt := 'Generic error code of the multi turn module is detected';
					12697:	sAxisErrTxt := 'Braking resistor overload';
					16512:	sAxisErrTxt	:= 'Drive overtemperature (IPM)';
					16513:	sAxisErrTxt	:= 'Drive overtemperature (controller)';
					16534:	sAxisErrTxt := 'Temperature sensor inoperative';
					17168:	sAxisErrTxt	:= 'Power stage overtemperature';
					17280:	sAxisErrTxt := 'The encoder temperature is too high';
					17424:	sAxisErrTxt	:= 'Motor overtemperature';
					21808:	sAxisErrTxt	:= 'System error detected (nonvolatilememory)';
					21893:	sAxisErrTxt	:= 'Error detected in non-volatile memory';
					21889:	sAxisErrTxt	:= 'System error detected (nonvolatile memory)';
					21890:	sAxisErrTxt	:= 'System error detected (CAN power supply)';
					21891:	sAxisErrTxt	:= 'System error detected (selftest)';
					21894:	sAxisErrTxt	:= 'System error detected (NV ACCESS)';
					25472:	sAxisErrTxt	:= 'Target position rejected';
					25985:	sAxisErrTxt	:= 'System error detected(FPGA)';
					28816:	sAxisErrTxt	:= 'System error detected (FPGA does NOT match firmware)';
					28817:	sAxisErrTxt	:= 'Emergency Stop Activated';
					28961:	sAxisErrTxt := 'Motor blocked';
					29080:	sAxisErrTxt := 'Commutation error detected';
					29568:  sAxisErrTxt	:= 'Error detected in communication with motor encoder';
					29574:	sAxisErrTxt	:= 'Drive is not synchronous wit master cycle';
					29581:	sAxisErrTxt := 'System error detected (encoder)';
					29587:	sAxisErrTxt	:= 'Encoder overvoltage or overcurrent';
					29592:	sAxisErrTxt := 'The returned position value are no longer considered valid';
					29593:	sAxisErrTxt := 'The multi turn encoder requires an explicit configuration command';
					30081:	sAxisErrTxt := 'Target position rejected';
					30082:	sAxisErrTxt := 'No target values received via the fieldbus';
					33072:	sAxisErrTxt	:= 'CANopen: Heartbeat error detected';
					33296:	sAxisErrTxt := 'R_PDO is too short';
					33921:	sAxisErrTxt	:= 'Actual Motor Velocity Too High';
					33553:	sAxisErrTxt	:= 'Motor torque too high FOR an excessive period OF time';
					33664:	sAxisErrTxt := 'Unstable current loop';
					33922:	sAxisErrTxt := 'Velocity deviation too high';
					34321:	sAxisErrTxt	:= 'Position deviation too high';
					34432:	sAxisErrTxt := 'Position deviation via signal output function MC_OK';
					34441:	sAxisErrTxt := 'Position deviation too high (following error)';
					61568:	sAxisErrTxt	:= 'Fieldbus: Communication	error detected';
					65282:	sAxisErrTxt	:= 'Not possible to read data of electronic motor nameplate';
					65296:	sAxisErrTxt	:= 'Forward Limit Switch Error';
					65297:	sAxisErrTxt	:= 'Reverse Limit Switch Error';
					65281:	sAxisErrTxt := 'System error detected';
					65298:	sAxisErrTxt	:= 'Forward Software Limit';
					65299:	sAxisErrTxt	:= 'Reverse Software Limit';
					65301:	sAxisErrTxt := 'The encoder firmware cannot operate on the provided hardware';

				END_CASE

			EstunPronet:
				CASE tyParamOut.udiAxisErrID OF
					65281:	sAxisErrTxt	:= 'Parameter breakdown';//A01
					65282:	sAxisErrTxt	:= 'AD shift channels breakdown';
					65283:	sAxisErrTxt	:= 'Overspeed';
					65284:	sAxisErrTxt	:= 'Overload';
					65285:	sAxisErrTxt := 'Position error counteroverflow ';
					65286:	sAxisErrTxt := 'Position error pulse overflow';
					65287:	sAxisErrTxt	:= 'The setting of electronic gear or given pulse frequency is not reasonable';
					65288:	sAxisErrTxt	:= 'The 1st channel of current detection is wrong.';
					65289:	sAxisErrTxt	:= 'The 2nd channel of current detection is wrong.';
					65290:	sAxisErrTxt	:= 'Incremental Encoder is break off.';//A10
					65292:	sAxisErrTxt	:= 'Overcurrent';
					65293:	sAxisErrTxt	:= 'Overvoltage';
					65294:	sAxisErrTxt	:= 'Undervoltage';
					65295:	sAxisErrTxt := 'Bleeder resistor error';
					65296:	sAxisErrTxt := 'Regeneration error';
					65297:	sAxisErrTxt := 'Resolver error';
					65298:	sAxisErrTxt := 'IGBT superheat alarm';
					65299:	sAxisErrTxt := 'Motor overheat alarm';
					65300:	sAxisErrTxt := 'Power line phase shortage';//A20
					65301:	sAxisErrTxt	:= 'Instantaneous power off alarm';
					65302:	sAxisErrTxt	:= 'Motor temperature detection sensor is break off.';
					65303:	sAxisErrTxt := 'Brake overcurrent alarm';//A23
					65305:	sAxisErrTxt := 'Motor power line U overcurrent';//A25
					65306:	sAxisErrTxt := 'Motor power line V overcurrent';//A26
					65307:	sAxisErrTxt := 'Motor power line W overcurrent';//A27
					65322:	sAxisErrTxt	:= 'Servomotor type error';//A42
					65323:	sAxisErrTxt	:= 'Servo drive type error';
					65325:	sAxisErrTxt	:= 'Absolute encoder multiturn information error';
					65326:	sAxisErrTxt	:= 'Absolute encoder multiturn information overflow';
					65327:	sAxisErrTxt	:= 'Battery voltage below 2.5V';
					65328:	sAxisErrTxt	:= 'Battery voltage below 3.1V';//A48
					65330:	sAxisErrTxt := 'Serial encoder communication overtime ';//A50
					65331:	sAxisErrTxt := 'Absolute encoder overspeed alarm detected';
					65332:  sAxisErrTxt	:= 'Absolute state of serial encoder error';
					65333:	sAxisErrTxt	:= 'Serial encoder calcaution error';
					65334:	sAxisErrTxt := 'Parity bit or end bit in serial encoder control domain error';
					65335:	sAxisErrTxt	:= 'Serial encoder communication data checking error';
					65336:	sAxisErrTxt := 'End bit in serial encoder control domain error';
					65338:	sAxisErrTxt := 'Serial encoder data empty';
					65339:	sAxisErrTxt := 'Serial encoder data format error';
					65340:	sAxisErrTxt := 'Communication module not detected ';//A60
					65341:	sAxisErrTxt := 'Communication unsuccessful';
					65342:	sAxisErrTxt := 'Servo drive can not receive the period data of communication module ';
					65343:	sAxisErrTxt := 'Communication module can not receive the servo drive response data.';
					65344:	sAxisErrTxt := 'Communication module and bus connectionless';
					65346:	sAxisErrTxt := 'CAN communication abnormal';
					65347:	sAxisErrTxt := 'Receiving heartbeat timeout';
					65349:	sAxisErrTxt := 'Synchronization signal monitoring cycle is longer than setting';
					65362: sAxisErrTxt	:= 'Torque output alarm';
				END_CASE
		END_CASE

	ELSE

		tyParamOut.bAxisErr			:= FALSE;
		tyParamOut.bFwdLmtSen		:= FALSE;
		tyParamOut.bInPos			:= FALSE;
		tyParamOut.bIsHomed			:= FALSE;
		tyParamOut.bPosDiff			:= TRUE;
		tyParamOut.bPwrOn			:= FALSE;
		tyParamOut.bRevLmtSen		:= FALSE;
		tyParamOut.bStopped			:= TRUE;
		tyParamOut.diActualPosInUM	:= 0;
		tyParamOut.diHmAcc			:= 0;
		tyParamOut.diHmSpdForSwitch	:= 0;
		tyParamOut.diHmSpdForZero	:= 0;
		tyParamOut.diProfileAcc		:= 0;
		tyParamOut.diProfileDec		:= 0;
		tyParamOut.udiAxisErrID		:= 0;

		bWidthPosDiff				:= TRUE;

	END_IF

	//Abnormal Movement
//	IF eStatus1 <> Error THEN
//		IF p_bOps = TRUE AND eStatus = Idle THEN
//			IF (ABS(tyParamOut.diActualPosInUM - diActualPosInUMOld) > 2000) AND (ABS(tyParamOut.diActualPosInUM - diActualPosInUMOld) < 10000) THEN
//				eStatus1	:= Error;
//				udiStatus1	:= 10000;	//Axis Move Abnormally By External Force
//
//				fMotionCANRstCtrlWord(ADR(tyParamOutDriver));
//				p_eAct	:= AWActIdle;
//				eStat	:= AWActIdle;
//			END_IF
//		ELSE
//			diActualPosInUMOld	:= tyParamOut.diActualPosInUM;
//		END_IF
//	END_IF

	//Reset Error
	IF (eStatus1 = Error) AND bRstErr THEN
		eStatus1	:= Idle;
		udiStatus1	:= 0;
	END_IF

	//Request Position To Movement Out Of Range
	IF p_bOps
		AND((tyParamInMove.diPosInUM < p_diMinAbsPosInUM) OR (tyParamInMove.diPosInUM > p_diMaxAbsPosInUM))
		AND (eStatus2 <> Error) THEN
		eStatus2	:= Error;
		udiStatus2	:= 10029;	//Request Absolute Position Out Of Range

		fMotionCANRstCtrlWord(ADR(tyParamOutDriver));
		p_eAct	:= AWActIdle;
		eStat	:= AWActIdle;
	END_IF

	//Reset Error
	IF (eStatus2 = Error) AND bRstErr THEN
		eStatus2	:= Idle;
		udiStatus2	:= 0;
	END_IF

	//Sensor Interrupt
	IF (bNotInterruptible = TRUE OR bJogging) AND eStatus3 <> Error THEN

		IF p_bInletSensor = TRUE THEN
			eStatus3	:= Error;
			udiStatus3	:= 10030;	//Inlet Sensor Interrupt Auto Width Movement

			fMotionCANRstCtrlWord(ADR(tyParamOutDriver));
			p_eAct	:= AWActIdle;
			eStat	:= AWActIdle;

		ELSIF p_bOutletSensor = TRUE THEN
			eStatus3	:= Error;
			udiStatus3	:= 10031;	//Outlet Sensor Interrupt Auto Width Movement

			fMotionCANRstCtrlWord(ADR(tyParamOutDriver));
			p_eAct	:= AWActIdle;
			eStat	:= AWActIdle;

		ELSIF p_bClearSensor = TRUE THEN
			eStatus3	:= Error;
			udiStatus3	:= 10032;	//Clear Sensor Interrupt Auto Width Movement

			fMotionCANRstCtrlWord(ADR(tyParamOutDriver));
			p_eAct	:= AWActIdle;
			eStat	:= AWActIdle;

		ELSIF p_bMiddleSensor = TRUE THEN
			eStatus3	:= Error;
			udiStatus3	:= 10033;	//Middle Sensor Interrupt Auto Width Movement

			fMotionCANRstCtrlWord(ADR(tyParamOutDriver));
			p_eAct	:= AWActIdle;
			eStat	:= AWActIdle;

		ELSIF p_bInterruptSensor = TRUE THEN
			eStatus3	:= Error;
			udiStatus3	:= 10034;	//Sensor Interrupt Auto Width Movement

			fMotionCANRstCtrlWord(ADR(tyParamOutDriver));
			p_eAct	:= AWActIdle;
			eStat	:= AWActIdle;

		ELSIF p_bCloseInterruptSensor = TRUE AND bJogOpen = FALSE THEN
			eStatus3	:= Error;
			udiStatus3	:= 10047;	//Sensor Interrupt Auto Width Movement

			fMotionCANRstCtrlWord(ADR(tyParamOutDriver));
			p_eAct	:= AWActIdle;
			eStat	:= AWActIdle;

		ELSIF p_bOpenInterruptSensor = TRUE AND bJogClose = FALSE THEN
			eStatus3	:= Error;
			udiStatus3	:= 10048;	//Sensor Interrupt Auto Width Movement

			fMotionCANRstCtrlWord(ADR(tyParamOutDriver));
			p_eAct	:= AWActIdle;
			eStat	:= AWActIdle;
		END_IF

	END_IF

	//Reset Error
	IF (eStatus3 = Error AND bRstErr)
		OR (p_bOpenInterruptSensor AND eStat = AWActJogClose)
		OR (p_bCloseInterruptSensor AND eStat = AWActJogOpen)
		THEN
		eStatus3	:= Idle;
		udiStatus3	:= 0;
	END_IF

	IF bRstErr THEN
		udiStatus	:= 0;
		bJogging	:= FALSE;
		bJogClose	:= FALSE;
		bJogOpen	:= FALSE;
	END_IF

	fbServoModuleOk(IN:= bModuleOK);
	fbServoModuleNotOk(IN:= bModuleOK = FALSE);
	IF fbServoModuleNotOk.Q AND udiStatus <> 10001 THEN

		bModuleNotOK		:= TRUE;
		bModuleNotOKLock	:= TRUE;
		usiRstStep	:= 0;
		tyParamOutDriver.uiCtrlword_6040	:= 0;
		tyParamOutDriver.siModOfOpt_6060	:= 0;
		tyParamOutDriver.diTargetPos_607A	:= 0;
		tyParamOutDriver.udiMoveSpd_6081	:= 0;
		tyParamOutDriver.siHmMethod_6098	:= 0;
		tyParamOutDriver.diJogVel_60FF		:= 0;

		CASE p_eNtParamMotorType OF

			DeltaAsdaA2:
				fbModuleOK(bModuleOK:= FALSE);
				IF eStatus = Idle THEN
					eAct	:= AWActRstNode;
				END_IF

				IF (eStatus = Done OR eStatus = Error)AND eStat = AWActRstNode THEN

					eAct	:= AWActIdle;
				END_IF

			EstunPronet:
				fbModuleOK(bModuleOK:= FALSE);
				IF eStatus = Idle THEN
					eAct	:= AWActRstNode;
				END_IF

				IF (eStatus = Done OR eStatus = Error)AND eStat = AWActRstNode THEN

					eAct	:= AWActIdle;
				END_IF

			SchneiderLexium28:
			// Do Nothing
		END_CASE

	ELSIF bModuleNotOK = TRUE AND fbServoModuleOk.Q THEN

		CASE usiRstStep OF

			0:
				IF eStatus = Idle THEN
					eAct	:= AWActRstAxisErr;
				END_IF

				IF eStatus = Done AND eStat = AWActRstAxisErr THEN
					eAct	:= AWActIdle;
					usiRstStep	:= 4;
				END_IF

			4: tyParamOutDriver.siModOfOpt_6060 := 1;
				usiRstStep	:= 5;

			5: tyParamOutDriver.siModOfOpt_6060 := 1;
				fbRstNodeTimer(IN:=TRUE);

				IF tyParamInDriver.siModOfOptDisp_6061 = 1 THEN
					usiRstStep	:= 6;
					fbRstNodeTimer(IN:=FALSE);
				ELSIF fbRstNodeTimer.Q THEN
					usiRstStep	:= 8;
					fbRstNodeTimer(IN:=FALSE);
				END_IF

			6: tyParamOutDriver.siModOfOpt_6060 := 6;
				fbRstNodeTimer(IN:=FALSE);
				usiRstStep	:= 7;

			7: tyParamOutDriver.siModOfOpt_6060 := 6;
				fbRstNodeTimer(IN:=TRUE);

				IF tyParamInDriver.siModOfOptDisp_6061 = 6 THEN
					usiRstStep	:= 10;
					fbRstNodeTimer(IN:=FALSE);
				ELSIF fbRstNodeTimer.Q THEN
					usiRstStep	:= 9;
					fbRstNodeTimer(IN:=FALSE);
				END_IF

			8:	fbModuleOK(bEn := TRUE, bModuleOK:= FALSE);
				fbRstNodeTimer(IN:=FALSE);
				usiRstStep	:= 9;

			9:	fbModuleOK(bModuleOK:= FALSE);
				IF eStatus = Idle THEN
					eAct	:=AWActRstNode;
				END_IF

				IF eStatus = Done AND eStat = AWActRstNode THEN
					usiRstStep	:= 0;
					eAct		:= AWActIdle;
				END_IF

			10:IF eStatus = Idle THEN
					eAct	:= AWActRstAxisErr;
				END_IF

				IF eStatus = Done AND eStat = AWActRstAxisErr THEN
					eAct			:=AWActIdle;
					usiRstStep	:= 11;
				END_IF

			11:

				IF eStatus = Idle THEN
					eAct	:= AWActSDOWrite;
				END_IF

				IF eStatus = Done AND eStat = AWActSDOWrite THEN
					eAct			:= AWActIdle;
					usiRstStep	:= 13;

				ELSIF udiStatus = 10028 THEN
					eAct			:= AWActIdle;
					usiRstStep	:= 0;
				END_IF

			13: bModuleNotOK	:= FALSE;
				usiRstStep	:= 0;
		END_CASE
	ELSE
		eAct	:= AWActIdle;

	END_IF

	IF tyParamOut.bPosDiff = FALSE THEN
		tyParamOutDriver.uiCtrlword_6040.4	:= FALSE;
	END_IF

END_ACTION
```

#### Act_InitGlobal.st
```iecst
(** 2019-04-09 **)
ACTION Act_InitGlobal:

	(* Always Change If Project Change *)

	//Pass Data To Link
	p_bLinkOpsRun ACCESS p_OpsRun;
	p_bLinkStartupRun ACCESS p_StartupRun;

	p_eLinkMag ACCESS p_NtParamProjMag;
	p_usiLinkMod ACCESS p_ProdRcpCurrRcp1McMod;
	p_eLinkTravAct ACCESS  p_OpsTravLifLDTravAct;
	p_bLinkSafetyRelay ACCESS p_DISafetyRlySig;
	p_bNtParamAutoRcpPrep ACCESS p_NtParamAutoRcpPrep;
	p_bHermesSvyPrep ACCESS p_NtParamHermesSvyPrep; //queryWO
	p_bMcParamHermesSvyEn ACCESS p_McParamHermesSvyEn;
	p_eNtParamCustomerReq ACCESS p_NtParamCustomerReq;
	p_bMcParamMesRFIDEn ACCESS p_McParamMesRFIDEn;

	//Pass Data To Internal Use
	p_udiRstErr ACCESS p_RstErrReset;
	p_bEn ACCESS p_DISimServoEn;
	p_bPrep ACCESS p_NtParamAWPrep;
	p_bDis ACCESS p_McParamAWDis;
	p_bOps ACCESS p_OpsStatusRun;
	p_bManual ACCESS p_UIMnlMod;
	p_diWidthAtHmPos ACCESS p_McParamWidthAtHmPos;
	p_tyTuning ACCESS p_NtParamAWTuning;
	p_diJogVelInUMPS ACCESS p_UIMnlAWJogSpd;
	p_diMovePosInUM ACCESS p_UIMnlAWTargetPos;
	p_diMoveDistInUM ACCESS p_UIMnlAWStepSize;
	p_bUITeachServo ACCESS p_UITeachServo;
	p_diMoveAcc ACCESS p_NtParamAWAcc;
	p_diMoveDec ACCESS p_NtParamAWDec;
	p_diMinWidthInUM ACCESS p_NtParamProdRcpMinWidth;
	p_diMaxWidthInUM ACCESS p_NtParamProdRcpMaxWidth;
	p_diWidthOffsetInUM ACCESS p_NtParamWidthOffset;
	p_bInletSensor ACCESS p_DIConvLftSen;
	p_bOutletSensor ACCESS p_DIConvRgtSen;
	p_bDir ACCESS p_NtParamAWDir;
	p_bDirBl ACCESS p_NtParamAWDirBl;
	p_usiNode ACCESS p_NtParamAWNode;
	p_sDevice ACCESS p_NtParamAWDevice;
	p_sProgNm ACCESS p_NtParamAWProgNm;
	p_diMoveBacklashDistInUM ACCESS p_NtParamAWMovBlDistInUM;
	p_diPitchInUM ACCESS p_NtParamAWPitchInUM;
	p_tyParamInHm ACCESS p_NtParamAWParamInHm;
	p_tyParamInConvert ACCESS p_NtParamAWParamInConvert;
	p_bNtSettingsLoadDone ACCESS p_StartupNtSettingsLoadDone;
	p_eNtParamMotorType ACCESS p_NtParamAWMotorType;

	p_bInletShutterCloseRS ACCESS p_DIInShutterCloseRS;
	p_bOutletShutterCloseRS ACCESS p_DIOutShutterCloseRS;
	p_bProjInletShutPrep ACCESS p_NtParamProjInletShutPrep;
//	p_bInShutterDis ACCESS p_McParamInShutterDis;
	p_bProjOutletShutPrep ACCESS p_NtParamProjOutletShutPrep;
	p_bOutShutterDis ACCESS p_McParamOutShutterDis;
	p_bPullerRetSen ACCESS p_DIPullerRetRS;
	p_bPullerExtSen ACCESS p_DIPullerExtRS;
	p_eTravLifPosGo ACCESS p_OpsTravLifLDPosGo;
	(* Always Change If Project Change *)

END_ACTION
```

#### Act_Link.st
```iecst
(** 2019-03-29 **)
ACTION Act_Link:

	IF p_bManual = TRUE THEN
		p_diGoWidth ACCESS p_UIMnlAWGoWidth;
		p_diMoveVelInUMPS ACCESS p_UIMnlAWNomSpd;
	ELSE
//		p_diGoWidth ACCESS p_ProdRcpCurrRcp2Width;
		p_diMoveVelInUMPS ACCESS p_NtParamAWAutoSpd;

		IF p_eLinkMag = LDMagQuadruple THEN
			CASE p_usiLinkMod OF
				0: //LDModLoadLnA:
					p_diGoWidth ACCESS p_ProdRcpCurrRcp2Width;

				1: //LDModLoadLnB:
					p_diGoWidth ACCESS p_ProdRcpCurrRcp2WidthRear;

				2: //LDModLoadLnAB:
//					IF p_eLinkTravAct = TravActGoAPos THEN
//						p_diGoWidth ACCESS p_ProdRcpCurrRcp2Width;
//					ELSIF p_eLinkTravAct = TravActGoBPos THEN
//						p_diGoWidth ACCESS p_ProdRcpCurrRcp2Width;
//					ELSIF p_eLinkTravAct = TravActGoCPos THEN
//						p_diGoWidth ACCESS p_ProdRcpCurrRcp2WidthRear;
//					ELSIF p_eLinkTravAct = TravActGoGPos THEN
//						p_diGoWidth ACCESS p_ProdRcpCurrRcp2WidthRear;
//					END_IF

					IF p_eTravLifPosGo = TravLifLDPosUS1 THEN
						p_diGoWidth ACCESS p_ProdRcpCurrRcp2Width;
					ELSIF p_eTravLifPosGo = TravLifLDPosUS2 THEN
						p_diGoWidth ACCESS p_ProdRcpCurrRcp2Width;
					ELSIF p_eTravLifPosGo = TravLifLDPosUS3 THEN
						p_diGoWidth ACCESS p_ProdRcpCurrRcp2WidthRear;
					ELSIF p_eTravLifPosGo = TravLifLDPosUS4 THEN
						p_diGoWidth ACCESS p_ProdRcpCurrRcp2WidthRear;
					END_IF
			END_CASE
		ELSE
			IF p_bNtParamAutoRcpPrep AND ((p_bHermesSvyPrep  AND p_bMcParamHermesSvyEn) OR (p_eNtParamCustomerReq = We_Fabricate AND p_bMcParamMesRFIDEn)) THEN
				p_diGoWidth ACCESS p_AutoRcpTravLifWidth;
			ELSE
				p_diGoWidth ACCESS p_ProdRcpCurrRcp2Width;
				//p_diGoWidth ACCESS ADR(diGoWidth);
			END_IF

		END_IF
	END_IF

	IF p_bProjInletShutPrep = TRUE THEN

		IF p_bInletShutterCloseRS = FALSE OR p_bPullerRetSen = FALSE OR p_bPullerExtSen
			THEN
			bInterruptSensor1 := TRUE;
		ELSE
			bInterruptSensor1 := FALSE;
		END_IF
	ELSE
		bInterruptSensor1 := FALSE;
	END_IF

	IF p_bProjOutletShutPrep = TRUE AND p_bOutShutterDis = FALSE THEN
		IF p_bOutletShutterCloseRS = FALSE OR p_bPullerRetSen = FALSE OR p_bPullerExtSen
			THEN
			bInterruptSensor2 := TRUE;
		ELSE
			bInterruptSensor2 := FALSE;
		END_IF
	ELSE
		bInterruptSensor2 := FALSE;
	END_IF

	p_bInterruptSensor := bInterruptSensor2 OR bInterruptSensor1;// OR p_bLinkSafetyRelay = FALSE;

END_ACTION
```

#### Act_LinkAction.st
```iecst
(** 2019-10-21 **)
ACTION Act_LinkAction:

	IF eStatus = Idle THEN
		IF bModuleNotOK THEN
			p_eAct ACCESS ADR(eAct);
		ELSE
			IF p_bLinkStartupRun = TRUE THEN
				p_eAct ACCESS p_StartupAWAct;
			ELSIF p_bLinkOpsRun = TRUE THEN
				p_eAct ACCESS p_OpsTravLifLDAWAct;
			ELSIF p_bManual = TRUE THEN
				p_eAct ACCESS p_UIAWOpenAct;
			ELSE
				p_eAct ACCESS ADR(eAct);
			END_IF
		END_IF
	END_IF

	IF EDGENEG(p_bManual) OR EDGENEG(p_bLinkOpsRun) OR EDGENEG(p_bLinkStartupRun) THEN
		tyParamOutDriver.uiCtrlword_6040	:= 0;
	END_IF

END_ACTION
```

### Program Logical/CANOpenServo/AW/AWPushOrPuller

#### InputRef.var
```iecst
(*2020-05-26*)
(**)
(*General*)
VAR
	p_eAct : REFERENCE TO eAWAction;
	p_udiRstErr : REFERENCE TO UDINT;
	p_bPrep : REFERENCE TO BOOL;
	p_bEn : REFERENCE TO BOOL;
	p_bDis : REFERENCE TO BOOL;
END_VAR
(**)
(*Configuration*)
VAR
	p_bOps : REFERENCE TO BOOL;
	p_bManual : REFERENCE TO BOOL;
	p_diWidthAtHmPos : REFERENCE TO DINT;
	p_tyTuning : REFERENCE TO tyMotionCANTuning;
	p_diGoWidth : REFERENCE TO DINT;
	p_diJogVelInUMPS : REFERENCE TO DINT;
	p_diMovePosInUM : REFERENCE TO DINT;
	p_diMoveDistInUM : REFERENCE TO DINT;
	p_diMoveVelInUMPS : REFERENCE TO DINT;
	p_diMoveAcc : REFERENCE TO DINT;
	p_diMoveDec : REFERENCE TO DINT;
	p_diMinAbsPosInUM : REFERENCE TO DINT;
	p_diMaxAbsPosInUM : REFERENCE TO DINT;
	p_diMinWidthInUM : REFERENCE TO DINT;
	p_diMaxWidthInUM : REFERENCE TO DINT;
	p_diWidthOffsetInUM : REFERENCE TO DINT;
	p_bInletSensor : REFERENCE TO BOOL;
	p_bOutletSensor : REFERENCE TO BOOL;
	p_bClearSensor : REFERENCE TO BOOL;
	p_bMiddleSensor : REFERENCE TO BOOL;
	p_bInterruptSensor : REFERENCE TO BOOL;
	p_bOpenInterruptSensor : REFERENCE TO BOOL;
	p_bCloseInterruptSensor : REFERENCE TO BOOL;
	p_bSafetyInterruptSen : REFERENCE TO BOOL;
	p_bDir : REFERENCE TO BOOL;
	p_bDirBl : REFERENCE TO BOOL;
	p_bNoIndexPulse : REFERENCE TO BOOL;
	p_usiNode : REFERENCE TO USINT;
	p_sDevice : REFERENCE TO STRING[3];
	p_sProgNm : REFERENCE TO STRING[15];
	p_diMoveBacklashDistInUM : REFERENCE TO DINT;
	p_diPitchInUM : REFERENCE TO DINT;
	p_tyParamInHm : REFERENCE TO tyMotionCANParamInHm;
	p_tyParamInConvert : REFERENCE TO tyMotionCANParamInConvert;
	p_bNtSettingsLoadDone : REFERENCE TO BOOL;
	p_eNtParamMotorType : REFERENCE TO eServoMotorType;
	p_bOutletShutterCloseRS : REFERENCE TO BOOL;
	p_bProjInletShutPrep : REFERENCE TO BOOL;
	p_bInShutterDis : REFERENCE TO BOOL;
	p_bOutShutterDis : REFERENCE TO BOOL;
	p_bProjOutletShutPrep : REFERENCE TO BOOL;
	p_bInletShutterCloseRS : REFERENCE TO BOOL;
	p_bUITeachServo : REFERENCE TO BOOL;
	p_bPullerExtSen : REFERENCE TO BOOL;
	p_bPullerRetSen : REFERENCE TO BOOL;
END_VAR
```
